KUKA KRL program: MyProgram_248().src

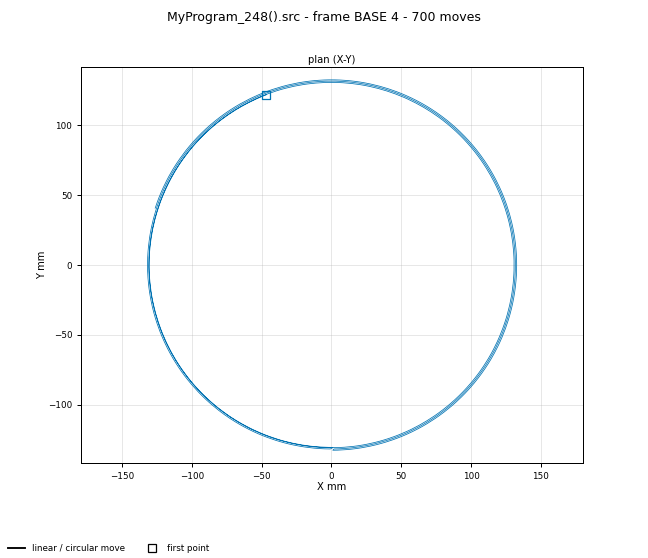
[picture p0: tool path of MyProgram_248().src in frame BASE 4, 700 of 700 moves have a stored position in this frame; points joined in program order, loops and branches not executed]
&ACCESS RVP
&REL 1
&PARAM TEMPLATE = C:\KRC\Roboter\Template\vorgabe
&PARAM EDITMASK = *
DEF MyProgram_248()
; ---- Setting reference (Base) ----
$BASE = BASE_DATA[4]

; --------------------------
; ---- Setting tool (TCP) ----
$TOOL = TOOL_DATA[3]
; --------------------------

$VEL.CP = VEL_APROX_PRINT
Startdeposition()
$VEL.CP = VEL_PRINT
LIN {X -46.6832,Y 121.9902,Z 163,A 110.8737,B 12.7153,C -0.1174,E1 12.6581,E2 699.2371} C_DIS
LIN {X -49.9782,Y 120.6763,Z 163,A 112.3319,B 12.7153,C -0.1132,E1 12.6544,E2 697.7915} C_DIS
LIN {X -53.5556,Y 119.1314,Z 163,A 114.1157,B 12.7153,C -0.1128,E1 12.6498,E2 696.0006} C_DIS
LIN {X -57.2848,Y 117.3848,Z 163,A 115.8599,B 12.7154,C -0.1089,E1 12.6454,E2 694.2652} C_DIS
LIN {X -59.7951,Y 116.1264,Z 163,A 117.1162,B 12.7154,C -0.1077,E1 12.6423,E2 693.0071} C_DIS
LIN {X -62.9383,Y 114.4547,Z 163,A 118.6303,B 12.7154,C -0.1043,E1 12.6386,E2 691.5001} C_DIS
LIN {X -65.207,Y 113.1772,Z 163,A 119.9528,B 12.7154,C -0.1069,E1 12.6353,E2 690.1578} C_DIS
LIN {X -68.5198,Y 111.2027,Z 163,A 121.5343,B 12.7154,C -0.1015,E1 12.6316,E2 688.5907} C_DIS
LIN {X -71.225,Y 109.4895,Z 163,A 122.9481,B 12.7155,C -0.0994,E1 12.6283,E2 687.1773} C_DIS
LIN {X -73.8707,Y 107.7222,Z 163,A 124.3516,B 12.7155,C -0.0972,E1 12.625,E2 685.7742} C_DIS
LIN {X -76.4904,Y 105.8783,Z 163,A 125.7574,B 12.7155,C -0.0947,E1 12.6218,E2 684.3698} C_DIS
LIN {X -79.0882,Y 103.9525,Z 163,A 127.1877,B 12.7155,C -0.0924,E1 12.6186,E2 682.9396} C_DIS
LIN {X -82.2352,Y 101.4811,Z 163,A 128.9913,B 12.7155,C -0.0902,E1 12.6147,E2 681.1323} C_DIS
LIN {X -85.3227,Y 98.8989,Z 163,A 130.775,B 12.7155,C -0.0871,E1 12.6109,E2 679.3484} C_DIS
LIN {X -88.3103,Y 96.2406,Z 163,A 132.6231,B 12.7156,C -0.0857,E1 12.607,E2 677.4913} C_DIS
LIN {X -91.2151,Y 93.4926,Z 163,A 134.4135,B 12.7156,C -0.0829,E1 12.6034,E2 675.6986} C_DIS
LIN {X -94.1515,Y 90.5351,Z 163,A 136.2687,B 12.7156,C -0.0795,E1 12.5998,E2 673.8423} C_DIS
LIN {X -97.2048,Y 87.2479,Z 163,A 138.1813,B 12.7156,C -0.0738,E1 12.5962,E2 671.9384} C_DIS
LIN {X -99.9408,Y 84.1001,Z 163,A 139.9545,B 12.7157,C -0.0683,E1 12.593,E2 670.1738} C_DIS
LIN {X -102.0114,Y 81.5764,Z 163,A 141.5514,B 12.7157,C -0.0687,E1 12.5902,E2 668.5594} C_DIS
LIN {X -104.7092,Y 78.083,Z 163,A 143.3581,B 12.7157,C -0.0611,E1 12.5872,E2 666.77} C_DIS
LIN {X -106.3801,Y 75.791,Z 163,A 144.7627,B 12.7157,C -0.0617,E1 12.5849,E2 665.3482} C_DIS
LIN {X -108.8838,Y 72.1487,Z 163,A 146.7321,B 12.7157,C -0.0576,E1 12.5818,E2 663.3776} C_DIS
LIN {X -111.0171,Y 68.8201,Z 163,A 148.3315,B 12.7157,C -0.05,E1 12.5794,E2 661.796} C_DIS
LIN {X -112.8395,Y 65.7903,Z 163,A 150.0583,B 12.7157,C -0.05,E1 12.5769,E2 660.0506} C_DIS
LIN {X -115.0342,Y 61.8715,Z 163,A 151.9693,B 12.7158,C -0.0435,E1 12.5744,E2 658.1488} C_DIS
LIN {X -116.6759,Y 58.7157,Z 163,A 153.4482,B 12.7158,C -0.0374,E1 12.5725,E2 656.6811} C_DIS
LIN {X -118.0782,Y 55.8412,Z 163,A 154.889,B 12.7158,C -0.0345,E1 12.5708,E2 655.2377} C_DIS
LIN {X -119.2704,Y 53.245,Z 163,A 156.2038,B 12.7158,C -0.0325,E1 12.5693,E2 653.9172} C_DIS
LIN {X -120.6709,Y 49.9913,Z 163,A 157.6764,B 12.7158,C -0.0263,E1 12.5677,E2 652.456} C_DIS
LIN {X -121.7339,Y 47.3425,Z 163,A 159.0481,B 12.7158,C -0.0256,E1 12.5663,E2 651.0717} C_DIS
LIN {X -122.9737,Y 44.023,Z 163,A 160.5652,B 12.7158,C -0.0203,E1 12.5648,E2 649.561} C_DIS
LIN {X -124.0232,Y 40.9732,Z 163,A 161.9931,B 12.7158,C -0.0166,E1 12.5635,E2 648.1332} C_DIS
LIN {X -124.9945,Y 37.9073,Z 163,A 163.4198,B 12.7158,C -0.0129,E1 12.5624,E2 646.7064} C_DIS
LIN {X -125.794,Y 35.1618,Z 163,A 164.7429,B 12.7158,C -0.0109,E1 12.5613,E2 645.3767} C_DIS
LIN {X -126.6177,Y 32.0694,Z 163,A 166.1098,B 12.7158,C -0.006,E1 12.5604,E2 644.0158} C_DIS
LIN {X -127.4419,Y 28.6231,Z 163,A 167.6781,B 12.7158,C -0.0018,E1 12.5594,E2 642.4477} C_DIS
LIN {X -128.0367,Y 25.8293,Z 163,A 168.986,B 12.7158,C 0.0007,E1 12.5587,E2 641.1349} C_DIS
LIN {X -128.6915,Y 22.3488,Z 163,A 170.4906,B 12.7158,C 0.0063,E1 12.5579,E2 639.6379} C_DIS
LIN {X -129.156,Y 19.4811,Z 163,A 171.8014,B 12.7158,C 0.0093,E1 12.5574,E2 638.3244} C_DIS
LIN {X -129.5892,Y 16.3576,Z 163,A 173.1987,B 12.7158,C 0.013,E1 12.5568,E2 636.927} C_DIS
LIN {X -129.9523,Y 13.1691,Z 163,A 174.7524,B 12.7158,C 0.0139,E1 12.5564,E2 635.3579} C_DIS
LIN {X -130.2342,Y 9.9928,Z 163,A 176.0604,B 12.7158,C 0.0201,E1 12.5561,E2 634.0621} C_DIS
LIN {X -130.4875,Y 5.8387,Z 163,A 178.0776,B 12.7158,C 0.0212,E1 12.5558,E2 632.0246} C_DIS
LIN {X -130.6007,Y 2.0177,Z 163,A 179.5385,B 12.7158,C 0.031,E1 12.5557,E2 630.5908} C_DIS
LIN {X -130.6106,Y -1.3842,Z 163,A -178.8919,B 12.7158,C 0.0337,E1 12.5557,E2 629.0138} C_DIS
LIN {X -130.52,Y -5.011,Z 163,A -177.2402,B 12.7158,C 0.037,E1 12.5559,E2 627.3568} C_DIS
LIN {X -130.3104,Y -8.9487,Z 163,A -175.3685,B 12.7158,C 0.0389,E1 12.5562,E2 625.4704} C_DIS
LIN {X -130.0173,Y -12.4916,Z 163,A -173.9505,B 12.7158,C 0.0467,E1 12.5565,E2 624.0706} C_DIS
LIN {X -129.633,Y -16.0033,Z 163,A -172.3925,B 12.7158,C 0.0511,E1 12.557,E2 622.5132} C_DIS
LIN {X -129.2325,Y -18.9667,Z 163,A -171.0719,B 12.7158,C 0.0547,E1 12.5575,E2 621.1929} C_DIS
LIN {X -128.8196,Y -21.5878,Z 163,A -169.825,B 12.7158,C 0.0562,E1 12.5581,E2 619.9375} C_DIS
LIN {X -128.1778,Y -25.1263,Z 163,A -168.2019,B 12.7158,C 0.0598,E1 12.559,E2 618.3106} C_DIS
LIN {X -127.5268,Y -28.2472,Z 163,A -166.7611,B 12.7158,C 0.0628,E1 12.5598,E2 616.8663} C_DIS
LIN {X -126.7017,Y -31.7385,Z 163,A -165.2684,B 12.7158,C 0.0692,E1 12.5608,E2 615.3846} C_DIS
LIN {X -125.9783,Y -34.5028,Z 163,A -164.042,B 12.7157,C 0.0733,E1 12.5617,E2 614.1626} C_DIS
LIN {X -125.0954,Y -37.5777,Z 163,A -162.5825,B 12.7157,C 0.076,E1 12.5628,E2 612.6978} C_DIS
LIN {X -124.1519,Y -40.5868,Z 163,A -161.1603,B 12.7157,C 0.079,E1 12.5641,E2 611.2723} C_DIS
LIN {X -123.0973,Y -43.6802,Z 163,A -159.7902,B 12.7157,C 0.0844,E1 12.5653,E2 609.9109} C_DIS
LIN {X -121.9894,Y -46.6852,Z 163,A -158.2103,B 12.7157,C 0.0842,E1 12.5669,E2 608.3117} C_DIS
LIN {X -120.672,Y -49.9886,Z 163,A -156.8729,B 12.7155,C 0.0936,E1 12.5683,E2 607.0018} C_DIS
LIN {X -119.4164,Y -52.9185,Z 163,A -155.3294,B 12.7155,C 0.0939,E1 12.57,E2 605.4423} C_DIS
LIN {X -118.2446,Y -55.4906,Z 163,A -153.9832,B 12.7155,C 0.0948,E1 12.5716,E2 604.0846} C_DIS
LIN {X -116.707,Y -58.6546,Z 163,A -152.5589,B 12.7155,C 0.1015,E1 12.5733,E2 602.6755} C_DIS
LIN {X -115.3567,Y -61.267,Z 163,A -151.1647,B 12.7155,C 0.1024,E1 12.5752,E2 601.27} C_DIS
LIN {X -113.82,Y -64.0779,Z 163,A -149.6509,B 12.7155,C 0.1034,E1 12.5772,E2 599.7444} C_DIS
LIN {X -111.5694,Y -67.9218,Z 163,A -147.6613,B 12.7155,C 0.1075,E1 12.5801,E2 597.7521} C_DIS
LIN {X -109.2975,Y -71.5202,Z 163,A -145.7821,B 12.7155,C 0.1117,E1 12.5829,E2 595.8727} C_DIS
LIN {X -106.7955,Y -75.2043,Z 163,A -144.0551,B 12.7153,C 0.1217,E1 12.5856,E2 594.1738} C_DIS
LIN {X -104.9142,Y -77.8076,Z 163,A -142.5374,B 12.7153,C 0.1224,E1 12.5881,E2 592.6441} C_DIS
LIN {X -103.0812,Y -80.2202,Z 163,A -141.1619,B 12.7153,C 0.1243,E1 12.5905,E2 591.2638} C_DIS
LIN {X -100.5659,Y -83.3513,Z 163,A -139.3096,B 12.7153,C 0.1261,E1 12.5938,E2 589.4018} C_DIS
LIN {X -97.7543,Y -86.6318,Z 163,A -137.3785,B 12.7153,C 0.1293,E1 12.5973,E2 587.4674} C_DIS
LIN {X -94.7689,Y -89.8884,Z 163,A -135.4961,B 12.7152,C 0.1347,E1 12.6009,E2 585.5926} C_DIS
LIN {X -91.916,Y -92.8033,Z 163,A -133.6849,B 12.7152,C 0.1377,E1 12.6045,E2 583.7796} C_DIS
LIN {X -88.9031,Y -95.6933,Z 163,A -131.769,B 12.7152,C 0.1393,E1 12.6084,E2 581.8544} C_DIS
LIN {X -85.9341,Y -98.3681,Z 163,A -130.0988,B 12.7151,C 0.1445,E1 12.6118,E2 580.1947} C_DIS
LIN {X -82.9209,Y -100.9217,Z 163,A -128.3556,B 12.7151,C 0.1474,E1 12.6156,E2 578.4509} C_DIS
LIN {X -79.8515,Y -103.367,Z 163,A -126.5261,B 12.7151,C 0.1477,E1 12.6196,E2 576.609} C_DIS
LIN {X -76.7991,Y -105.6545,Z 163,A -124.9687,B 12.715,C 0.1533,E1 12.6231,E2 575.0658} C_DIS
LIN {X -74.4284,Y -107.3378,Z 163,A -123.6386,B 12.715,C 0.154,E1 12.6262,E2 573.7295} C_DIS
LIN {X -72.0249,Y -108.9652,Z 163,A -122.2836,B 12.715,C 0.154,E1 12.6293,E2 572.3651} C_DIS
LIN {X -68.8174,Y -111.0188,Z 163,A -120.7144,B 12.715,C 0.1589,E1 12.633,E2 570.8084} C_DIS
LIN {X -66.0644,Y -112.6786,Z 163,A -119.3006,B 12.7149,C 0.1608,E1 12.6364,E2 569.3943} C_DIS
LIN {X -63.6337,Y -114.0696,Z 163,A -117.9724,B 12.7149,C 0.16,E1 12.6397,E2 568.0544} C_DIS
LIN {X -60.1614,Y -115.9372,Z 163,A -116.3208,B 12.7149,C 0.1641,E1 12.6437,E2 566.4122} C_DIS
LIN {X -57.6106,Y -117.2241,Z 163,A -115.0672,B 12.7149,C 0.1656,E1 12.6469,E2 565.1586} C_DIS
LIN {X -54.7716,Y -118.577,Z 163,A -113.6686,B 12.7149,C 0.1667,E1 12.6504,E2 563.7578} C_DIS
LIN {X -51.4577,Y -120.053,Z 163,A -112.082,B 12.7148,C 0.1685,E1 12.6545,E2 562.1718} C_DIS
LIN {X -48.8184,Y -121.1496,Z 163,A -110.8254,B 12.7148,C 0.1697,E1 12.6577,E2 560.9148} C_DIS
LIN {X -45.5127,Y -122.4302,Z 163,A -109.264,B 12.7148,C 0.171,E1 12.6618,E2 559.3526} C_DIS
LIN {X -42.4978,Y -123.5091,Z 163,A -107.8552,B 12.7148,C 0.172,E1 12.6655,E2 557.9432} C_DIS
LIN {X -39.4561,Y -124.5142,Z 163,A -106.4463,B 12.7148,C 0.1731,E1 12.6692,E2 556.5337} C_DIS
LIN {X -36.7579,Y -125.3369,Z 163,A -105.1944,B 12.7148,C 0.1736,E1 12.6726,E2 555.2799} C_DIS
LIN {X -33.3,Y -126.3002,Z 163,A -103.6737,B 12.7147,C 0.176,E1 12.6767,E2 553.7654} C_DIS
LIN {X -30.2058,Y -127.0759,Z 163,A -102.2279,B 12.7147,C 0.1756,E1 12.6806,E2 552.3137} C_DIS
LIN {X -27.1009,Y -127.7743,Z 163,A -100.8642,B 12.7147,C 0.1771,E1 12.6843,E2 550.9536} C_DIS
LIN {X -24.1906,Y -128.3567,Z 163,A -99.5117,B 12.7147,C 0.1763,E1 12.6881,E2 549.5946} C_DIS
LIN {X -21.085,Y -128.9035,Z 163,A -98.0994,B 12.7147,C 0.1761,E1 12.692,E2 548.1785} C_DIS
LIN {X -17.9213,Y -129.3819,Z 163,A -96.7699,B 12.7147,C 0.1784,E1 12.6956,E2 546.8575} C_DIS
LIN {X -14.7423,Y -129.7835,Z 163,A -95.212,B 12.7147,C 0.1747,E1 12.7,E2 545.2808} C_DIS
LIN {X -11.214,Y -130.134,Z 163,A -93.8584,B 12.7147,C 0.1802,E1 12.7037,E2 543.9507} C_DIS
LIN {X -8.366,Y -130.3483,Z 163,A -92.4343,B 12.7147,C 0.1758,E1 12.7077,E2 542.5055} C_DIS
LIN {X -5.153,Y -130.5145,Z 163,A -91.1022,B 12.7147,C 0.1779,E1 12.7114,E2 541.1823} C_DIS
LIN {X -1.9527,Y -130.6018,Z 163,A -89.6778,B 12.7147,C 0.1772,E1 12.7154,E2 539.7549} C_DIS
LIN {X 0.9174,Y -130.6131,Z 163,A -88.8333,B 12.7145,C 0.188,E1 12.7176,E2 538.9595} C_DIS
Enddeposition()
LIN {X 0.9174,Y -130.6131,Z 163,A -88.8333,B 12.7145,C 0.188,E1 12.7176,E2 538.9595} C_DIS
Startdeposition()
$VEL.CP = VEL_PRINT
LIN {X 2.9572,Y -130.8103,Z 164,A -87.5272,B 12.7129,C 0.1767,E1 12.7196,E2 537.6024} C_DIS
LIN {X 6.1659,Y -130.6972,Z 164,A -86.0767,B 12.7129,C 0.1751,E1 12.7236,E2 536.1458} C_DIS
LIN {X 9.3838,Y -130.505,Z 164,A -84.7313,B 12.7129,C 0.1764,E1 12.7274,E2 534.8076} C_DIS
LIN {X 12.8176,Y -130.2129,Z 164,A -83.2362,B 12.7129,C 0.1762,E1 12.7315,E2 533.3133} C_DIS
LIN {X 15.6281,Y -129.9052,Z 164,A -81.9766,B 12.7129,C 0.175,E1 12.735,E2 532.0504} C_DIS
LIN {X 18.9476,Y -129.4633,Z 164,A -80.5189,B 12.7129,C 0.1744,E1 12.739,E2 530.5928} C_DIS
LIN {X 22.132,Y -128.9577,Z 164,A -79.0774,B 12.7129,C 0.1727,E1 12.743,E2 529.1468} C_DIS
LIN {X 25.5213,Y -128.3298,Z 164,A -77.6997,B 12.7129,C 0.1753,E1 12.7468,E2 527.784} C_DIS
LIN {X 28.6831,Y -127.6598,Z 164,A -76.2844,B 12.7129,C 0.1742,E1 12.7506,E2 526.3676} C_DIS
LIN {X 30.9937,Y -127.1182,Z 164,A -75.149,B 12.7129,C 0.1707,E1 12.7538,E2 525.2199} C_DIS
LIN {X 34.8731,Y -126.1092,Z 164,A -73.5047,B 12.7129,C 0.1721,E1 12.7582,E2 523.5877} C_DIS
LIN {X 37.9309,Y -125.2234,Z 164,A -72.07,B 12.7129,C 0.1697,E1 12.762,E2 522.147} C_DIS
LIN {X 41.2594,Y -124.1659,Z 164,A -70.4025,B 12.713,C 0.1643,E1 12.7665,E2 520.4615} C_DIS
LIN {X 45.586,Y -122.6438,Z 164,A -68.5096,B 12.713,C 0.1652,E1 12.7714,E2 518.5809} C_DIS
LIN {X 48.3557,Y -121.5795,Z 164,A -67.2192,B 12.713,C 0.1639,E1 12.7748,E2 517.2906} C_DIS
LIN {X 51.5406,Y -120.2631,Z 164,A -65.8052,B 12.713,C 0.1646,E1 12.7784,E2 515.8866} C_DIS
LIN {X 54.2495,Y -119.0672,Z 164,A -64.4511,B 12.713,C 0.1612,E1 12.7819,E2 514.5245} C_DIS
LIN {X 57.1852,Y -117.6857,Z 164,A -63.0198,B 12.713,C 0.1589,E1 12.7855,E2 513.0907} C_DIS
LIN {X 60.261,Y -116.1399,Z 164,A -61.5367,B 12.7131,C 0.1574,E1 12.7892,E2 511.609} C_DIS
LIN {X 62.8821,Y -114.7428,Z 164,A -60.1838,B 12.7131,C 0.1539,E1 12.7925,E2 510.2486} C_DIS
LIN {X 65.678,Y -113.1654,Z 164,A -58.8716,B 12.7131,C 0.1543,E1 12.7957,E2 508.9464} C_DIS
LIN {X 68.4316,Y -111.5218,Z 164,A -57.43,B 12.7131,C 0.1509,E1 12.7991,E2 507.4988} C_DIS
LIN {X 71.1439,Y -109.8114,Z 164,A -56.0328,B 12.7132,C 0.1487,E1 12.8024,E2 506.101} C_DIS
LIN {X 73.8295,Y -108.0243,Z 164,A -54.6378,B 12.7132,C 0.1467,E1 12.8056,E2 504.7068} C_DIS
LIN {X 76.4534,Y -106.1839,Z 164,A -53.1819,B 12.7132,C 0.1427,E1 12.809,E2 503.2431} C_DIS
LIN {X 79.7631,Y -103.7205,Z 164,A -51.426,B 12.7132,C 0.1407,E1 12.8129,E2 501.4913} C_DIS
LIN {X 82.9013,Y -101.2293,Z 164,A -49.6993,B 12.7133,C 0.138,E1 12.8166,E2 499.7662} C_DIS
LIN {X 85.3739,Y -99.1528,Z 164,A -48.2801,B 12.7133,C 0.135,E1 12.8197,E2 498.3448} C_DIS
LIN {X 88.3689,Y -96.4934,Z 164,A -46.5394,B 12.7133,C 0.1317,E1 12.8233,E2 496.6037} C_DIS
LIN {X 91.3657,Y -93.6612,Z 164,A -44.7492,B 12.7134,C 0.1283,E1 12.8269,E2 494.8134} C_DIS
LIN {X 94.2093,Y -90.8002,Z 164,A -42.8838,B 12.7134,C 0.1215,E1 12.8305,E2 492.9339} C_DIS
LIN {X 97.0246,Y -87.7852,Z 164,A -41.0985,B 12.7135,C 0.118,E1 12.8339,E2 491.1491} C_DIS
LIN {X 100.0304,Y -84.3446,Z 164,A -39.2261,B 12.7135,C 0.117,E1 12.8373,E2 489.2899} C_DIS
LIN {X 102.5806,Y -81.2238,Z 164,A -37.4588,B 12.7135,C 0.1127,E1 12.8404,E2 487.5203} C_DIS
LIN {X 105.0905,Y -77.9488,Z 164,A -35.7098,B 12.7135,C 0.11,E1 12.8433,E2 485.776} C_DIS
LIN {X 106.8866,Y -75.4668,Z 164,A -34.3578,B 12.7136,C 0.1063,E1 12.8455,E2 484.4212} C_DIS
LIN {X 108.7849,Y -72.7038,Z 164,A -32.9309,B 12.7136,C 0.1038,E1 12.8478,E2 482.9975} C_DIS
LIN {X 110.5434,Y -70.0013,Z 164,A -31.5399,B 12.7136,C 0.1008,E1 12.8499,E2 481.6073} C_DIS
LIN {X 112.2262,Y -67.2709,Z 164,A -29.9994,B 12.7137,C 0.0932,E1 12.8521,E2 480.0487} C_DIS
LIN {X 114.5187,Y -63.2888,Z 164,A -28.1177,B 12.7137,C 0.0917,E1 12.8547,E2 478.1804} C_DIS
LIN {X 116.0276,Y -60.4749,Z 164,A -26.7681,B 12.7137,C 0.0893,E1 12.8564,E2 476.8349} C_DIS
LIN {X 117.5747,Y -57.4102,Z 164,A -25.2801,B 12.7137,C 0.0857,E1 12.8583,E2 475.3468} C_DIS
LIN {X 118.8392,Y -54.7426,Z 164,A -23.9675,B 12.7138,C 0.0815,E1 12.8598,E2 474.0303} C_DIS
LIN {X 120.259,Y -51.5502,Z 164,A -22.5189,B 12.7138,C 0.0797,E1 12.8614,E2 472.5896} C_DIS
LIN {X 121.4863,Y -48.5868,Z 164,A -21.1028,B 12.7138,C 0.0754,E1 12.8629,E2 471.1704} C_DIS
LIN {X 122.5606,Y -45.8082,Z 164,A -19.7787,B 12.7138,C 0.0712,E1 12.8642,E2 469.8424} C_DIS
LIN {X 123.9688,Y -41.8512,Z 164,A -17.8515,B 12.7139,C 0.0633,E1 12.866,E2 467.9023} C_DIS
LIN {X 125.1387,Y -38.2075,Z 164,A -16.3407,B 12.7139,C 0.0633,E1 12.8673,E2 466.4094} C_DIS
LIN {X 126.1006,Y -34.9037,Z 164,A -14.8825,B 12.7139,C 0.0605,E1 12.8684,E2 464.9552} C_DIS
LIN {X 126.9173,Y -31.807,Z 164,A -13.468,B 12.7139,C 0.056,E1 12.8694,E2 463.5376} C_DIS
LIN {X 127.6574,Y -28.6936,Z 164,A -12.1068,B 12.7139,C 0.0531,E1 12.8702,E2 462.1795} C_DIS
LIN {X 128.3029,Y -25.6535,Z 164,A -10.7502,B 12.7139,C 0.0492,E1 12.871,E2 460.8218} C_DIS
LIN {X 128.8767,Y -22.5953,Z 164,A -9.3815,B 12.7139,C 0.045,E1 12.8717,E2 459.4507} C_DIS
LIN {X 129.3921,Y -19.4319,Z 164,A -7.9572,B 12.7139,C 0.0403,E1 12.8723,E2 458.0224} C_DIS
LIN {X 129.8586,Y -16.0182,Z 164,A -6.4988,B 12.714,C 0.0373,E1 12.8728,E2 456.5682} C_DIS
LIN {X 130.1891,Y -13.0648,Z 164,A -5.212,B 12.714,C 0.0339,E1 12.8732,E2 455.2816} C_DIS
LIN {X 130.487,Y -9.63,Z 164,A -3.7393,B 12.714,C 0.0305,E1 12.8735,E2 453.8116} C_DIS
LIN {X 130.6726,Y -6.6548,Z 164,A -2.4043,B 12.714,C 0.0257,E1 12.8737,E2 452.4715} C_DIS
LIN {X 130.7933,Y -3.5686,Z 164,A -1.0691,B 12.714,C 0.0222,E1 12.8738,E2 451.1369} C_DIS
LIN {X 130.8438,Y -0.0051,Z 164,A 0.3845,B 12.714,C 0.0207,E1 12.8738,E2 449.6944} C_DIS
LIN {X 130.81,Y 2.965,Z 164,A 1.7444,B 12.714,C 0.0151,E1 12.8738,E2 448.3259} C_DIS
LIN {X 130.7112,Y 5.8858,Z 164,A 3.1328,B 12.714,C 0.0081,E1 12.8736,E2 446.9232} C_DIS
LIN {X 130.5047,Y 9.3874,Z 164,A 4.5066,B 12.714,C 0.0083,E1 12.8734,E2 445.5671} C_DIS
LIN {X 130.2123,Y 12.8233,Z 164,A 5.9871,B 12.714,C 0.0047,E1 12.873,E2 444.0885} C_DIS
LIN {X 129.8877,Y 15.7743,Z 164,A 7.2744,B 12.714,C 0.0013,E1 12.8726,E2 442.8013} C_DIS
LIN {X 129.4605,Y 18.9672,Z 164,A 8.6844,B 12.714,C -0.0028,E1 12.872,E2 441.3899} C_DIS
LIN {X 128.9575,Y 22.1333,Z 164,A 10.0542,B 12.714,C -0.0059,E1 12.8714,E2 440.0228} C_DIS
LIN {X 128.3296,Y 25.5223,Z 164,A 11.4734,B 12.714,C -0.0077,E1 12.8707,E2 438.6127} C_DIS
LIN {X 127.6647,Y 28.6616,Z 164,A 12.8714,B 12.714,C -0.0115,E1 12.8698,E2 437.2142} C_DIS
LIN {X 127.1257,Y 30.9627,Z 164,A 14.0476,B 12.714,C -0.0186,E1 12.8691,E2 436.0201} C_DIS
LIN {X 126.1183,Y 34.8406,Z 164,A 15.5966,B 12.714,C -0.0176,E1 12.868,E2 434.4939} C_DIS
LIN {X 125.2532,Y 37.8335,Z 164,A 17.002,B 12.714,C -0.0226,E1 12.8668,E2 433.0824} C_DIS
LIN {X 124.4586,Y 40.372,Z 164,A 18.3592,B 12.714,C -0.0315,E1 12.8657,E2 431.7012} C_DIS
LIN {X 123.194,Y 44.0777,Z 164,A 19.896,B 12.714,C -0.0311,E1 12.8643,E2 430.184} C_DIS
LIN {X 122.0769,Y 47.0833,Z 164,A 21.2033,B 12.714,C -0.0321,E1 12.863,E2 428.887} C_DIS
LIN {X 120.9801,Y 49.8367,Z 164,A 22.5072,B 12.714,C -0.0358,E1 12.8616,E2 427.5813} C_DIS
LIN {X 119.7152,Y 52.8035,Z 164,A 23.9618,B 12.714,C -0.0409,E1 12.86,E2 426.1206} C_DIS
LIN {X 118.4142,Y 55.6615,Z 164,A 25.3445,B 12.714,C -0.0447,E1 12.8584,E2 424.7359} C_DIS
LIN {X 116.9748,Y 58.6262,Z 164,A 26.8279,B 12.714,C -0.0497,E1 12.8565,E2 423.2465} C_DIS
LIN {X 115.3941,Y 61.6787,Z 164,A 28.1997,B 12.714,C -0.0497,E1 12.8548,E2 421.8894} C_DIS
LIN {X 114.0584,Y 64.1144,Z 164,A 29.4816,B 12.714,C -0.0547,E1 12.853,E2 420.5988} C_DIS
LIN {X 112.3615,Y 67.044,Z 164,A 30.9152,B 12.714,C -0.057,E1 12.851,E2 419.1699} C_DIS
LIN {X 110.8493,Y 69.5166,Z 164,A 32.2505,B 12.714,C -0.0621,E1 12.849,E2 417.8259} C_DIS
LIN {X 108.9256,Y 72.493,Z 164,A 33.7051,B 12.714,C -0.0631,E1 12.8468,E2 416.3818} C_DIS
LIN {X 107.1096,Y 75.1506,Z 164,A 35.0977,B 12.7139,C -0.066,E1 12.8446,E2 414.9902} C_DIS
LIN {X 105.0942,Y 77.9439,Z 164,A 36.7258,B 12.7139,C -0.0729,E1 12.8419,E2 413.3471} C_DIS
LIN {X 102.6588,Y 81.1252,Z 164,A 38.4806,B 12.7139,C -0.0769,E1 12.8389,E2 411.5912} C_DIS
LIN {X 100.2025,Y 84.1395,Z 164,A 40.0666,B 12.7139,C -0.0774,E1 12.836,E2 410.0181} C_DIS
LIN {X 97.4808,Y 87.2782,Z 164,A 41.9544,B 12.7138,C -0.0833,E1 12.8325,E2 408.1212} C_DIS
LIN {X 94.7615,Y 90.2236,Z 164,A 43.696,B 12.7138,C -0.0866,E1 12.8292,E2 406.3804} C_DIS
LIN {X 91.9519,Y 93.0858,Z 164,A 45.4537,B 12.7138,C -0.0903,E1 12.8257,E2 404.6217} C_DIS
LIN {X 88.9689,Y 95.9406,Z 164,A 47.2429,B 12.7138,C -0.0933,E1 12.8221,E2 402.834} C_DIS
LIN {X 85.7549,Y 98.8241,Z 164,A 49.0357,B 12.7138,C -0.0942,E1 12.8184,E2 401.0521} C_DIS
LIN {X 82.9996,Y 101.149,Z 164,A 50.6759,B 12.7137,C -0.0988,E1 12.8148,E2 399.404} C_DIS
LIN {X 79.7682,Y 103.7166,Z 164,A 52.4795,B 12.7137,C -0.1019,E1 12.8109,E2 397.6004} C_DIS
LIN {X 76.6517,Y 106.0402,Z 164,A 54.0346,B 12.7137,C -0.1007,E1 12.8074,E2 396.0621} C_DIS
LIN {X 74.0284,Y 107.8878,Z 164,A 55.3783,B 12.7137,C -0.1013,E1 12.8043,E2 394.7252} C_DIS
LIN {X 71.3742,Y 109.6619,Z 164,A 56.8102,B 12.7137,C -0.1044,E1 12.801,E2 393.289} C_DIS
LIN {X 68.6418,Y 111.3928,Z 164,A 58.2207,B 12.7137,C -0.1064,E1 12.7976,E2 391.8789} C_DIS
LIN {X 65.8901,Y 113.0426,Z 164,A 59.6239,B 12.7137,C -0.1084,E1 12.7943,E2 390.4758} C_DIS
LIN {X 63.2961,Y 114.5146,Z 164,A 60.9593,B 12.7136,C -0.111,E1 12.791,E2 389.1367} C_DIS
LIN {X 60.4719,Y 116.0292,Z 164,A 62.3206,B 12.7136,C -0.1117,E1 12.7877,E2 387.7801} C_DIS
LIN {X 57.3978,Y 117.5808,Z 164,A 63.7226,B 12.7136,C -0.1107,E1 12.7842,E2 386.3904} C_DIS
LIN {X 54.7508,Y 118.8354,Z 164,A 65.1214,B 12.7136,C -0.1154,E1 12.7806,E2 384.9779} C_DIS
LIN {X 51.8699,Y 120.1207,Z 164,A 66.4869,B 12.7136,C -0.1165,E1 12.7771,E2 383.6143} C_DIS
LIN {X 48.5905,Y 121.4848,Z 164,A 68.0197,B 12.7136,C -0.1176,E1 12.7732,E2 382.0842} C_DIS
LIN {X 45.8111,Y 122.5595,Z 164,A 69.3167,B 12.7136,C -0.1186,E1 12.7698,E2 380.7881} C_DIS
LIN {X 42.7934,Y 123.6456,Z 164,A 70.7158,B 12.7136,C -0.1198,E1 12.7661,E2 379.3898} C_DIS
LIN {X 39.7502,Y 124.6572,Z 164,A 72.115,B 12.7135,C -0.1209,E1 12.7624,E2 377.9913} C_DIS
LIN {X 36.6835,Y 125.5939,Z 164,A 73.5501,B 12.7135,C -0.1228,E1 12.7585,E2 376.5528} C_DIS
LIN {X 33.5741,Y 126.4607,Z 164,A 74.9551,B 12.7135,C -0.1235,E1 12.7547,E2 375.1489} C_DIS
LIN {X 30.241,Y 127.2996,Z 164,A 76.4213,B 12.7135,C -0.1235,E1 12.7508,E2 373.6877} C_DIS
LIN {X 27.3545,Y 127.9505,Z 164,A 77.6363,B 12.7135,C -0.1221,E1 12.7475,E2 372.4823} C_DIS
LIN {X 24.1889,Y 128.5869,Z 164,A 79.1239,B 12.7135,C -0.1247,E1 12.7434,E2 370.9864} C_DIS
LIN {X 20.7945,Y 129.1809,Z 164,A 80.6212,B 12.7135,C -0.125,E1 12.7393,E2 369.4911} C_DIS
LIN {X 17.6069,Y 129.6532,Z 164,A 82.0569,B 12.7135,C -0.1262,E1 12.7353,E2 368.0529} C_DIS
LIN {X 14.4223,Y 130.0452,Z 164,A 83.3824,B 12.7135,C -0.1245,E1 12.7316,E2 366.737} C_DIS
LIN {X 11.4698,Y 130.3389,Z 164,A 84.8155,B 12.7135,C -0.1283,E1 12.7276,E2 365.2889} C_DIS
LIN {X 8.2902,Y 130.5792,Z 164,A 86.1529,B 12.7135,C -0.1269,E1 12.7239,E2 363.9589} C_DIS
LIN {X 5.0188,Y 130.7457,Z 164,A 87.5978,B 12.7135,C -0.1273,E1 12.7199,E2 362.5133} C_DIS
LIN {X 1.6085,Y 130.8333,Z 164,A 89.0368,B 12.7135,C -0.1258,E1 12.7159,E2 361.0814} C_DIS
LIN {X -1.5992,Y 130.8335,Z 164,A 90.4132,B 12.7135,C -0.125,E1 12.7121,E2 359.709} C_DIS
LIN {X -4.5697,Y 130.7632,Z 164,A 91.7931,B 12.7135,C -0.1268,E1 12.7082,E2 358.3206} C_DIS
LIN {X -8.0118,Y 130.5964,Z 164,A 93.1603,B 12.7135,C -0.1229,E1 12.7044,E2 356.9706} C_DIS
LIN {X -10.9858,Y 130.3798,Z 164,A 94.6327,B 12.7135,C -0.1267,E1 12.7003,E2 355.4796} C_DIS
LIN {X -14.4179,Y 130.0457,Z 164,A 96.0767,B 12.7135,C -0.1245,E1 12.6963,E2 354.0441} C_DIS
LIN {X -17.363,Y 129.6851,Z 164,A 97.4026,B 12.7135,C -0.1245,E1 12.6926,E2 352.7159} C_DIS
LIN {X -20.3979,Y 129.2425,Z 164,A 98.7623,B 12.7135,C -0.1243,E1 12.6888,E2 351.3551} C_DIS
LIN {X -23.9457,Y 128.6334,Z 164,A 100.3542,B 12.7135,C -0.1237,E1 12.6845,E2 349.7625} C_DIS
LIN {X -26.8902,Y 128.0508,Z 164,A 101.7345,B 12.7135,C -0.1245,E1 12.6807,E2 348.3755} C_DIS
LIN {X -30.0123,Y 127.3548,Z 164,A 103.0636,B 12.7135,C -0.1217,E1 12.6771,E2 347.0557} C_DIS
LIN {X -33.1186,Y 126.5822,Z 164,A 104.539,B 12.7135,C -0.1224,E1 12.6731,E2 345.5727} C_DIS
LIN {X -36.2059,Y 125.7338,Z 164,A 105.944,B 12.7135,C -0.1212,E1 12.6693,E2 344.1683} C_DIS
LIN {X -39.5018,Y 124.7366,Z 164,A 107.3859,B 12.7135,C -0.1182,E1 12.6655,E2 342.7353} C_DIS
LIN {X -42.5426,Y 123.7325,Z 164,A 108.7995,B 12.7135,C -0.1171,E1 12.6617,E2 341.3215} C_DIS
LIN {X -45.4393,Y 122.6988,Z 164,A 110.1922,B 12.7135,C -0.1167,E1 12.6581,E2 339.9246} C_DIS
LIN {X -48.3601,Y 121.5777,Z 164,A 111.5195,B 12.7135,C -0.1141,E1 12.6546,E2 338.6035} C_DIS
LIN {X -51.1469,Y 120.4329,Z 164,A 112.9042,B 12.7135,C -0.1141,E1 12.651,E2 337.2122} C_DIS
LIN {X -54.2864,Y 119.0501,Z 164,A 114.4294,B 12.7135,C -0.1127,E1 12.6472,E2 335.6857} C_DIS
LIN {X -57.1797,Y 117.6884,Z 164,A 115.7611,B 12.7135,C -0.1092,E1 12.6438,E2 334.3633} C_DIS
LIN {X -60.2505,Y 116.1454,Z 164,A 117.2562,B 12.7136,C -0.1068,E1 12.6401,E2 332.8706} C_DIS
LIN {X -62.8599,Y 114.7548,Z 164,A 118.6178,B 12.7136,C -0.1065,E1 12.6368,E2 331.5026} C_DIS
LIN {X -65.6417,Y 113.1864,Z 164,A 119.9905,B 12.7136,C -0.1037,E1 12.6334,E2 330.1342} C_DIS
LIN {X -68.3777,Y 111.5548,Z 164,A 121.2822,B 12.7136,C -0.099,E1 12.6304,E2 328.8558} C_DIS
LIN {X -70.7876,Y 110.0417,Z 164,A 122.7415,B 12.7136,C -0.1021,E1 12.6269,E2 327.373} C_DIS
LIN {X -73.8298,Y 108.0241,Z 164,A 124.2531,B 12.7136,C -0.0973,E1 12.6234,E2 325.8731} C_DIS
LIN {X -76.453,Y 106.1842,Z 164,A 125.7318,B 12.7136,C -0.0966,E1 12.62,E2 324.387} C_DIS
LIN {X -79.7555,Y 103.7264,Z 164,A 127.5115,B 12.7137,C -0.0927,E1 12.6161,E2 322.6119} C_DIS
LIN {X -82.9065,Y 101.2251,Z 164,A 129.2696,B 12.7137,C -0.0892,E1 12.6123,E2 320.8561} C_DIS
LIN {X -85.3748,Y 99.152,Z 164,A 130.7112,B 12.7137,C -0.0871,E1 12.6092,E2 319.4126} C_DIS
LIN {X -88.3717,Y 96.4908,Z 164,A 132.5101,B 12.7137,C -0.0846,E1 12.6054,E2 317.6104} C_DIS
LIN {X -91.3716,Y 93.6554,Z 164,A 134.3068,B 12.7138,C -0.0805,E1 12.6018,E2 315.817} C_DIS
LIN {X -94.2095,Y 90.8,Z 164,A 136.2019,B 12.7138,C -0.0798,E1 12.5981,E2 313.9085} C_DIS
LIN {X -96.9464,Y 87.8713,Z 164,A 137.964,B 12.7138,C -0.076,E1 12.5948,E2 312.1476} C_DIS
LIN {X -99.7376,Y 84.69,Z 164,A 139.8101,B 12.7138,C -0.0716,E1 12.5914,E2 310.3044} C_DIS
LIN {X -102.5815,Y 81.2227,Z 164,A 141.7301,B 12.7138,C -0.0659,E1 12.5881,E2 308.3918} C_DIS
LIN {X -105.0931,Y 77.9454,Z 164,A 143.5149,B 12.7139,C -0.061,E1 12.5851,E2 306.6119} C_DIS
LIN {X -106.9728,Y 75.3447,Z 164,A 144.9031,B 12.7139,C -0.0572,E1 12.5828,E2 305.2272} C_DIS
LIN {X -108.7823,Y 72.7076,Z 164,A 146.3363,B 12.7139,C -0.0544,E1 12.5806,E2 303.7919} C_DIS
LIN {X -110.5227,Y 70.0341,Z 164,A 147.7441,B 12.7139,C -0.0511,E1 12.5785,E2 302.3846} C_DIS
LIN {X -112.1704,Y 67.3643,Z 164,A 149.144,B 12.7139,C -0.0482,E1 12.5764,E2 300.9833} C_DIS
LIN {X -113.7026,Y 64.7435,Z 164,A 150.5001,B 12.7139,C -0.0453,E1 12.5745,E2 299.6257} C_DIS
LIN {X -115.3943,Y 61.6784,Z 164,A 152.0503,B 12.7139,C -0.0416,E1 12.5725,E2 298.0753} C_DIS
LIN {X -116.7622,Y 59.0439,Z 164,A 153.3811,B 12.714,C -0.0389,E1 12.5708,E2 296.7424} C_DIS
LIN {X -118.1682,Y 56.1766,Z 164,A 154.7719,B 12.714,C -0.0349,E1 12.5691,E2 295.3542} C_DIS
LIN {X -119.6142,Y 53.0293,Z 164,A 156.3032,B 12.714,C -0.0311,E1 12.5673,E2 293.823} C_DIS
LIN {X -120.7829,Y 50.3089,Z 164,A 157.7452,B 12.714,C -0.0308,E1 12.5658,E2 292.3656} C_DIS
LIN {X -122.5626,Y 45.8029,Z 164,A 159.7582,B 12.714,C -0.0224,E1 12.5637,E2 290.3678} C_DIS
LIN {X -123.6484,Y 42.7852,Z 164,A 161.1784,B 12.714,C -0.0188,E1 12.5624,E2 288.9475} C_DIS
LIN {X -124.66,Y 39.7415,Z 164,A 162.5992,B 12.714,C -0.0152,E1 12.5612,E2 287.5264} C_DIS
LIN {X -125.5974,Y 36.6719,Z 164,A 164.0562,B 12.714,C -0.0123,E1 12.56,E2 286.0652} C_DIS
LIN {X -126.458,Y 33.5846,Z 164,A 165.4741,B 12.714,C -0.0086,E1 12.559,E2 284.6472} C_DIS
LIN {X -127.2991,Y 30.2431,Z 164,A 166.9646,B 12.714,C -0.0038,E1 12.558,E2 283.1608} C_DIS
LIN {X -127.9567,Y 27.3258,Z 164,A 168.314,B 12.714,C -0.0009,E1 12.5572,E2 281.8082} C_DIS
LIN {X -128.5869,Y 24.189,Z 164,A 169.7055,B 12.714,C 0.0035,E1 12.5565,E2 280.4194} C_DIS
LIN {X -129.179,Y 20.8059,Z 164,A 171.2185,B 12.714,C 0.0077,E1 12.5558,E2 278.9072} C_DIS
LIN {X -129.6483,Y 17.6436,Z 164,A 172.6627,B 12.714,C 0.0108,E1 12.5552,E2 277.4595} C_DIS
LIN {X -130.0398,Y 14.4725,Z 164,A 173.9868,B 12.714,C 0.0167,E1 12.5548,E2 276.1457} C_DIS
LIN {X -130.3401,Y 11.4558,Z 164,A 175.4781,B 12.714,C 0.0169,E1 12.5544,E2 274.6368} C_DIS
LIN {X -130.5958,Y 8.0206,Z 164,A 176.8894,B 12.714,C 0.0235,E1 12.5541,E2 273.2386} C_DIS
LIN {X -130.7333,Y 5.3344,Z 164,A 178.2219,B 12.714,C 0.0235,E1 12.5539,E2 271.8894} C_DIS
LIN {X -130.8333,Y 1.6097,Z 164,A 179.7634,B 12.714,C 0.0304,E1 12.5539,E2 270.3603} C_DIS
LIN {X -130.8372,Y -1.2667,Z 164,A -178.929,B 12.714,C 0.0331,E1 12.5539,E2 269.0485} C_DIS
LIN {X -130.7627,Y -4.5829,Z 164,A -177.4579,B 12.714,C 0.0369,E1 12.5539,E2 267.5767} C_DIS
LIN {X -130.5956,Y -8.0243,Z 164,A -175.9946,B 12.714,C 0.0424,E1 12.5542,E2 266.1204} C_DIS
LIN {X -130.3797,Y -10.9875,Z 164,A -174.5916,B 12.714,C 0.044,E1 12.5545,E2 264.7068} C_DIS
LIN {X -129.9621,Y -15.1508,Z 164,A -172.6626,B 12.714,C 0.0471,E1 12.5551,E2 262.7684} C_DIS
LIN {X -129.4928,Y -18.7415,Z 164,A -171.1847,B 12.714,C 0.0542,E1 12.5557,E2 261.3048} C_DIS
LIN {X -128.9572,Y -22.1353,Z 164,A -169.6034,B 12.714,C 0.0569,E1 12.5564,E2 259.7161} C_DIS
LIN {X -128.3319,Y -25.511,Z 164,A -168.2089,B 12.714,C 0.0637,E1 12.5571,E2 258.3359} C_DIS
LIN {X -127.6632,Y -28.6684,Z 164,A -166.776,B 12.7139,C 0.0673,E1 12.558,E2 256.9021} C_DIS
LIN {X -127.0764,Y -31.1671,Z 164,A -165.4907,B 12.7139,C 0.0668,E1 12.5588,E2 255.5989} C_DIS
LIN {X -126.1056,Y -34.886,Z 164,A -163.9346,B 12.7139,C 0.0745,E1 12.5599,E2 254.0594} C_DIS
LIN {X -125.2134,Y -37.9634,Z 164,A -162.4283,B 12.7139,C 0.0761,E1 12.5611,E2 252.5422} C_DIS
LIN {X -124.2387,Y -41.0408,Z 164,A -161.0053,B 12.7139,C 0.0798,E1 12.5624,E2 251.1194} C_DIS
LIN {X -123.195,Y -44.0747,Z 164,A -159.4472,B 12.7139,C 0.0802,E1 12.5638,E2 249.5445} C_DIS
LIN {X -121.5814,Y -48.351,Z 164,A -157.5592,B 12.7138,C 0.0883,E1 12.5657,E2 247.6717} C_DIS
LIN {X -120.2957,Y -51.4653,Z 164,A -156.122,B 12.7138,C 0.0931,E1 12.5673,E2 246.2402} C_DIS
LIN {X -119.129,Y -54.1141,Z 164,A -154.6778,B 12.7138,C 0.0924,E1 12.5689,E2 244.7762} C_DIS
LIN {X -117.7013,Y -57.1535,Z 164,A -153.2962,B 12.7137,C 0.0983,E1 12.5706,E2 243.4063} C_DIS
LIN {X -116.1429,Y -60.2553,Z 164,A -151.7892,B 12.7137,C 0.1025,E1 12.5725,E2 241.902} C_DIS
LIN {X -114.7474,Y -62.8735,Z 164,A -150.4554,B 12.7137,C 0.1051,E1 12.5743,E2 240.565} C_DIS
LIN {X -113.1728,Y -65.6652,Z 164,A -149.0327,B 12.7137,C 0.1081,E1 12.5762,E2 239.1412} C_DIS
LIN {X -111.5185,Y -68.437,Z 164,A -147.6589,B 12.7136,C 0.1126,E1 12.5782,E2 237.773} C_DIS
LIN {X -109.8039,Y -71.1554,Z 164,A -146.2156,B 12.7136,C 0.1152,E1 12.5804,E2 236.3265} C_DIS
LIN {X -108.033,Y -73.8169,Z 164,A -144.7787,B 12.7136,C 0.1176,E1 12.5827,E2 234.8861} C_DIS
LIN {X -106.1827,Y -76.4551,Z 164,A -143.2884,B 12.7136,C 0.1191,E1 12.5851,E2 233.3873} C_DIS
LIN {X -103.719,Y -79.7651,Z 164,A -141.502,B 12.7135,C 0.1237,E1 12.5881,E2 231.6044} C_DIS
LIN {X -101.2262,Y -82.9051,Z 164,A -139.7193,B 12.7135,C 0.127,E1 12.5912,E2 229.8196} C_DIS
LIN {X -99.0964,Y -85.4394,Z 164,A -138.1648,B 12.7135,C 0.1276,E1 12.594,E2 228.2533} C_DIS
LIN {X -96.4834,Y -88.3798,Z 164,A -136.4232,B 12.7134,C 0.1308,E1 12.5973,E2 226.5104} C_DIS
LIN {X -93.6505,Y -91.3766,Z 164,A -134.7034,B 12.7134,C 0.1366,E1 12.6006,E2 224.8017} C_DIS
LIN {X -90.8049,Y -94.2047,Z 164,A -132.8165,B 12.7134,C 0.1369,E1 12.6044,E2 222.9} C_DIS
LIN {X -87.8941,Y -96.9258,Z 164,A -131.0652,B 12.7133,C 0.1401,E1 12.608,E2 221.1487} C_DIS
LIN {X -84.8891,Y -99.5684,Z 164,A -129.2949,B 12.7133,C 0.1429,E1 12.6118,E2 219.3769} C_DIS
LIN {X -81.375,Y -102.4603,Z 164,A -127.3522,B 12.7133,C 0.1476,E1 12.616,E2 217.4408} C_DIS
LIN {X -77.9488,Y -105.0905,Z 164,A -125.5387,B 12.7132,C 0.1527,E1 12.62,E2 215.6372} C_DIS
LIN {X -75.3444,Y -106.973,Z 164,A -124.2261,B 12.7132,C 0.1573,E1 12.6229,E2 214.3362} C_DIS
LIN {X -72.7082,Y -108.7819,Z 164,A -122.6948,B 12.7132,C 0.1563,E1 12.6265,E2 212.7896} C_DIS
LIN {X -70.0066,Y -110.5401,Z 164,A -121.3278,B 12.7131,C 0.1595,E1 12.6297,E2 211.4282} C_DIS
LIN {X -67.2626,Y -112.2312,Z 164,A -119.8627,B 12.7131,C 0.1602,E1 12.6332,E2 209.957} C_DIS
LIN {X -64.4931,Y -113.8454,Z 164,A -118.5362,B 12.7131,C 0.164,E1 12.6364,E2 208.6398} C_DIS
LIN {X -61.6846,Y -115.391,Z 164,A -117.0164,B 12.7131,C 0.1629,E1 12.6402,E2 207.1064} C_DIS
LIN {X -59.0438,Y -116.7622,Z 164,A -115.6978,B 12.7131,C 0.1641,E1 12.6435,E2 205.786} C_DIS
LIN {X -55.9743,Y -118.2648,Z 164,A -114.2436,B 12.713,C 0.1669,E1 12.6471,E2 204.3369} C_DIS
LIN {X -53.0262,Y -119.6156,Z 164,A -112.7917,B 12.713,C 0.1677,E1 12.6508,E2 202.8812} C_DIS
LIN {X -50.289,Y -120.7912,Z 164,A -111.4498,B 12.713,C 0.1681,E1 12.6543,E2 201.5347} C_DIS
LIN {X -47.0915,Y -122.0737,Z 164,A -109.9068,B 12.713,C 0.1687,E1 12.6583,E2 199.9876} C_DIS
LIN {X -42.7971,Y -123.6443,Z 164,A -107.9606,B 12.713,C 0.1718,E1 12.6634,E2 198.048} C_DIS
LIN {X -39.7542,Y -124.656,Z 164,A -106.5523,B 12.713,C 0.1728,E1 12.6671,E2 196.6391} C_DIS
LIN {X -36.8335,Y -125.55,Z 164,A -105.1425,B 12.713,C 0.172,E1 12.6709,E2 195.2204} C_DIS
LIN {X -33.5864,Y -126.4575,Z 164,A -103.6988,B 12.7129,C 0.1737,E1 12.6748,E2 193.7804} C_DIS
LIN {X -30.6402,Y -127.2034,Z 164,A -102.4447,B 12.7129,C 0.1765,E1 12.6782,E2 192.5353} C_DIS
LIN {X -27.3368,Y -127.9544,Z 164,A -100.8887,B 12.7129,C 0.1754,E1 12.6825,E2 190.9702} C_DIS
LIN {X -24.1914,Y -128.5864,Z 164,A -99.508,B 12.7129,C 0.1766,E1 12.6862,E2 189.5921} C_DIS
LIN {X -21.3588,Y -129.0867,Z 164,A -98.2058,B 12.7129,C 0.1759,E1 12.6898,E2 188.2843} C_DIS
LIN {X -17.6092,Y -129.6528,Z 164,A -96.5667,B 12.7129,C 0.177,E1 12.6944,E2 186.6474} C_DIS
LIN {X -14.4274,Y -130.0447,Z 164,A -95.2389,B 12.7129,C 0.1793,E1 12.698,E2 185.3282} C_DIS
LIN {X -12.0331,Y -130.2882,Z 164,A -93.9449,B 12.7129,C 0.1731,E1 12.7017,E2 184.0049} C_DIS
LIN {X -8.0322,Y -130.5951,Z 164,A -92.4067,B 12.7129,C 0.179,E1 12.7059,E2 182.4923} C_DIS
LIN {X -4.8179,Y -130.7535,Z 164,A -90.9638,B 12.7129,C 0.1781,E1 12.71,E2 181.0448} C_DIS
LIN {X -1.61,Y -130.8333,Z 164,A -89.5811,B 12.7129,C 0.1786,E1 12.7138,E2 179.6642} C_DIS
LIN {X 0.9495,Y -130.8386,Z 164,A -88.9402,B 12.7126,C 0.1911,E1 12.7155,E2 179.0803} C_DIS
Enddeposition()
LIN {X 0.9495,Y -130.8386,Z 164,A -88.9402,B 12.7126,C 0.1911,E1 12.7155,E2 179.0803} C_DIS
Startdeposition()
$VEL.CP = VEL_PRINT
LIN {X -0.8075,Y -131.7592,Z 164,A -89.8661,B 12.7124,C 0.2033,E1 12.7127,E2 180.0615} C_DIS
LIN {X -4.6265,Y -131.6813,Z 164,A -91.4447,B 12.7124,C 0.2012,E1 12.7083,E2 181.6309} C_DIS
LIN {X -8.2381,Y -131.5038,Z 164,A -93.0669,B 12.7124,C 0.2025,E1 12.7037,E2 183.2597} C_DIS
LIN {X -12.4266,Y -131.1743,Z 164,A -94.9434,B 12.7124,C 0.2035,E1 12.6985,E2 185.1428} C_DIS
LIN {X -16.1659,Y -130.7672,Z 164,A -96.4621,B 12.7124,C 0.2002,E1 12.6943,E2 186.6481} C_DIS
LIN {X -18.8446,Y -130.407,Z 164,A -97.6685,B 12.7124,C 0.2007,E1 12.691,E2 187.8586} C_DIS
LIN {X -22.6401,Y -129.803,Z 164,A -99.4853,B 12.7124,C 0.2038,E1 12.6859,E2 189.6933} C_DIS
LIN {X -27.1004,Y -128.9462,Z 164,A -101.2817,B 12.7125,C 0.1984,E1 12.6811,E2 191.4689} C_DIS
LIN {X -30.5085,Y -128.1811,Z 164,A -103.1696,B 12.7124,C 0.207,E1 12.6758,E2 193.4012} C_DIS
LIN {X -33.7048,Y -127.3777,Z 164,A -104.3553,B 12.7124,C 0.1998,E1 12.6727,E2 194.5576} C_DIS
LIN {X -36.9587,Y -126.4716,Z 164,A -106.0636,B 12.7124,C 0.2049,E1 12.668,E2 196.2947} C_DIS
LIN {X -40.0547,Y -125.5254,Z 164,A -107.1928,B 12.7125,C 0.1967,E1 12.6651,E2 197.3908} C_DIS
LIN {X -43.4676,Y -124.3852,Z 164,A -108.7302,B 12.7125,C 0.1947,E1 12.661,E2 198.9251} C_DIS
LIN {X -46.2348,Y -123.3829,Z 164,A -110.1303,B 12.7125,C 0.1966,E1 12.6573,E2 200.3397} C_DIS
LIN {X -49.7648,Y -122.003,Z 164,A -111.6604,B 12.7125,C 0.1921,E1 12.6534,E2 201.8558} C_DIS
LIN {X -52.5482,Y -120.8294,Z 164,A -113.1042,B 12.7125,C 0.194,E1 12.6497,E2 203.3151} C_DIS
LIN {X -55.9205,Y -119.3077,Z 164,A -115.0636,B 12.7125,C 0.2009,E1 12.6446,E2 205.3161} C_DIS
LIN {X -59.4187,Y -117.6033,Z 164,A -116.1453,B 12.7127,C 0.1837,E1 12.6421,E2 206.3251} C_DIS
LIN {X -62.779,Y -115.8465,Z 164,A -117.9377,B 12.7127,C 0.1852,E1 12.6376,E2 208.1346} C_DIS
LIN {X -65.922,Y -114.0868,Z 164,A -119.4901,B 12.7127,C 0.1827,E1 12.6338,E2 209.6851} C_DIS
LIN {X -69.1526,Y -112.1584,Z 164,A -121.3451,B 12.7127,C 0.1858,E1 12.6294,E2 211.5659} C_DIS
LIN {X -73.0217,Y -109.6784,Z 164,A -123.3633,B 12.7127,C 0.1832,E1 12.6246,E2 213.586} C_DIS
LIN {X -76.9596,Y -106.9526,Z 164,A -125.5176,B 12.7127,C 0.1816,E1 12.6197,E2 215.7483} C_DIS
LIN {X -80.8358,Y -104.0532,Z 164,A -128.4954,B 12.7125,C 0.199,E1 12.6129,E2 218.828} C_DIS
LIN {X -86.3791,Y -99.5,Z 164,A -130.6286,B 12.7129,C 0.1698,E1 12.6086,E2 220.8442} C_DIS
LIN {X -89.6224,Y -96.5886,Z 164,A -132.4353,B 12.7129,C 0.164,E1 12.6049,E2 222.6396} C_DIS
LIN {X -92.3231,Y -94.0103,Z 164,A -134.1954,B 12.7129,C 0.164,E1 12.6013,E2 224.4153} C_DIS
LIN {X -95.507,Y -90.7746,Z 164,A -137.1768,B 12.7127,C 0.1838,E1 12.5954,E2 227.5139} C_DIS
LIN {X -100.2868,Y -85.4638,Z 164,A -139.146,B 12.7132,C 0.1504,E1 12.592,E2 229.3481} C_DIS
LIN {X -102.6912,Y -82.5594,Z 164,A -140.8197,B 12.7132,C 0.1475,E1 12.5891,E2 231.0248} C_DIS
LIN {X -104.7637,Y -79.9129,Z 164,A -142.4804,B 12.7132,C 0.1489,E1 12.5862,E2 232.7082} C_DIS
LIN {X -107.4272,Y -76.2958,Z 164,A -144.5312,B 12.7132,C 0.1467,E1 12.5828,E2 234.7693} C_DIS
LIN {X -109.4535,Y -73.3586,Z 164,A -146.0305,B 12.7132,C 0.1417,E1 12.5805,E2 236.2615} C_DIS
LIN {X -112.0686,Y -69.2983,Z 164,A -147.9472,B 12.7133,C 0.1323,E1 12.5776,E2 238.1551} C_DIS
LIN {X -113.5512,Y -66.8404,Z 164,A -149.3854,B 12.7133,C 0.1336,E1 12.5756,E2 239.6147} C_DIS
LIN {X -115.8215,Y -62.8248,Z 164,A -151.474,B 12.7133,C 0.1305,E1 12.5727,E2 241.7116} C_DIS
LIN {X -117.5363,Y -59.5504,Z 164,A -152.9177,B 12.7134,C 0.1225,E1 12.5709,E2 243.1348} C_DIS
LIN {X -119.7849,Y -54.8886,Z 164,A -155.2233,B 12.7134,C 0.1179,E1 12.5681,E2 245.445} C_DIS
LIN {X -121.6231,Y -50.6835,Z 164,A -157.2002,B 12.7135,C 0.1121,E1 12.566,E2 247.418} C_DIS
LIN {X -122.8223,Y -47.7039,Z 164,A -158.691,B 12.7135,C 0.1105,E1 12.5644,E2 248.9187} C_DIS
LIN {X -124.05,Y -44.4147,Z 164,A -160.1784,B 12.7135,C 0.1054,E1 12.563,E2 250.4001} C_DIS
LIN {X -125.0385,Y -41.5497,Z 164,A -161.5088,B 12.7136,C 0.102,E1 12.5618,E2 251.7307} C_DIS
LIN {X -126.1126,Y -38.1678,Z 164,A -163.3228,B 12.7136,C 0.1039,E1 12.5603,E2 253.5751} C_DIS
LIN {X -127.1901,Y -34.4083,Z 164,A -164.8903,B 12.7136,C 0.096,E1 12.5591,E2 255.1255} C_DIS
LIN {X -128.2826,Y -30.0863,Z 164,A -166.8966,B 12.7136,C 0.092,E1 12.5578,E2 257.1379} C_DIS
LIN {X -129.5208,Y -24.2015,Z 164,A -169.3901,B 12.7138,C 0.0817,E1 12.5564,E2 259.6145} C_DIS
LIN {X -130.2891,Y -19.6486,Z 164,A -171.8196,B 12.7138,C 0.0854,E1 12.5553,E2 262.0911} C_DIS
LIN {X -130.777,Y -16.084,Z 164,A -172.8813,B 12.7138,C 0.0695,E1 12.555,E2 263.0925} C_DIS
LIN {X -131.1306,Y -12.8815,Z 164,A -174.4476,B 12.7138,C 0.0691,E1 12.5545,E2 264.6767} C_DIS
LIN {X -131.4456,Y -9.1301,Z 164,A -176.2271,B 12.7138,C 0.0675,E1 12.5541,E2 266.4711} C_DIS
LIN {X -131.6911,Y -4.361,Z 164,A -178.1988,B 12.7138,C 0.059,E1 12.5539,E2 268.4283} C_DIS
LIN {X -131.7597,Y -0.7296,Z 164,A -179.8551,B 12.7139,C 0.056,E1 12.5539,E2 270.0918} C_DIS
LIN {X -131.7296,Y 2.9796,Z 164,A 178.6181,B 12.7139,C 0.0493,E1 12.5539,E2 271.6068} C_DIS
LIN {X -131.6404,Y 5.6756,Z 164,A 177.3532,B 12.7139,C 0.0479,E1 12.554,E2 272.8811} C_DIS
LIN {X -131.4291,Y 9.3564,Z 164,A 175.7374,B 12.7139,C 0.0434,E1 12.5543,E2 274.4965} C_DIS
LIN {X -131.1474,Y 12.7061,Z 164,A 174.238,B 12.7139,C 0.0399,E1 12.5547,E2 275.9986} C_DIS
LIN {X -130.3286,Y 19.3933,Z 164,A 171.3419,B 12.7139,C 0.0306,E1 12.5557,E2 278.8875} C_DIS
LIN {X -129.6738,Y 23.3617,Z 164,A 169.5387,B 12.7139,C 0.0266,E1 12.5566,E2 280.6949} C_DIS
LIN {X -128.9037,Y 27.2973,Z 164,A 167.4588,B 12.7139,C 0.0291,E1 12.5578,E2 282.8117} C_DIS
LIN {X -128.188,Y 30.4801,Z 164,A 166.5122,B 12.714,C 0.0143,E1 12.5583,E2 283.7018} C_DIS
LIN {X -127.5975,Y 32.865,Z 164,A 165.3038,B 12.714,C 0.0143,E1 12.5592,E2 284.9252} C_DIS
LIN {X -126.853,Y 35.628,Z 164,A 164.0273,B 12.714,C 0.0115,E1 12.5601,E2 286.2039} C_DIS
LIN {X -125.9469,Y 38.7093,Z 164,A 162.5376,B 12.714,C 0.0096,E1 12.5613,E2 287.7029} C_DIS
LIN {X -124.8774,Y 42.0336,Z 164,A 160.9234,B 12.714,C 0.0075,E1 12.5627,E2 289.3263} C_DIS
LIN {X -123.3174,Y 46.4097,Z 164,A 159.0015,B 12.714,C -0.0005,E1 12.5646,E2 291.2344} C_DIS
LIN {X -121.8399,Y 50.1642,Z 164,A 156.9693,B 12.714,C 0.001,E1 12.5667,E2 293.2966} C_DIS
LIN {X -120.0349,Y 54.341,Z 164,A 155.236,B 12.714,C -0.01,E1 12.5686,E2 294.9991} C_DIS
LIN {X -118.0879,Y 58.4487,Z 164,A 153.2402,B 12.714,C -0.015,E1 12.5711,E2 296.9947} C_DIS
LIN {X -116.2613,Y 62.0078,Z 164,A 151.3307,B 12.714,C -0.0157,E1 12.5735,E2 298.9219} C_DIS
LIN {X -114.1256,Y 65.8549,Z 164,A 148.5657,B 12.714,C -0.0014,E1 12.5776,E2 301.7823} C_DIS
LIN {X -110.6665,Y 71.5157,Z 164,A 146.6844,B 12.714,C -0.0316,E1 12.5802,E2 303.545} C_DIS
LIN {X -109.2147,Y 73.7134,Z 164,A 145.1685,B 12.714,C -0.026,E1 12.5826,E2 305.1024} C_DIS
LIN {X -107.3766,Y 76.3666,Z 164,A 143.9255,B 12.714,C -0.0331,E1 12.5846,E2 306.3252} C_DIS
LIN {X -104.9173,Y 79.7121,Z 164,A 142.0936,B 12.714,C -0.0369,E1 12.5876,E2 308.1581} C_DIS
LIN {X -102.1221,Y 83.2621,Z 164,A 140.1377,B 12.714,C -0.0417,E1 12.591,E2 310.1106} C_DIS
LIN {X -99.3879,Y 86.5076,Z 164,A 138.2881,B 12.714,C -0.0459,E1 12.5944,E2 311.9587} C_DIS
LIN {X -96.4364,Y 89.7859,Z 164,A 136.3487,B 12.714,C -0.0497,E1 12.5981,E2 313.8982} C_DIS
LIN {X -93.238,Y 93.1036,Z 164,A 134.2963,B 12.714,C -0.0529,E1 12.6021,E2 315.954} C_DIS
LIN {X -90.0555,Y 96.1853,Z 164,A 132.3457,B 12.714,C -0.0564,E1 12.606,E2 317.9053} C_DIS
LIN {X -86.7967,Y 99.1356,Z 164,A 130.4336,B 12.7139,C -0.0603,E1 12.61,E2 319.8154} C_DIS
LIN {X -83.4045,Y 102.0057,Z 164,A 128.5148,B 12.7139,C -0.0644,E1 12.6141,E2 321.7306} C_DIS
LIN {X -80.1268,Y 104.6001,Z 164,A 126.6838,B 12.7139,C -0.0675,E1 12.6181,E2 323.5612} C_DIS
LIN {X -76.775,Y 107.0846,Z 164,A 124.8483,B 12.7139,C -0.0703,E1 12.6223,E2 325.3972} C_DIS
LIN {X -73.3421,Y 109.4645,Z 164,A 123.0039,B 12.7139,C -0.0727,E1 12.6266,E2 327.243} C_DIS
LIN {X -69.629,Y 111.8628,Z 164,A 121.0945,B 12.7139,C -0.0762,E1 12.631,E2 329.149} C_DIS
LIN {X -63.863,Y 115.2519,Z 164,A 118.3844,B 12.7137,C -0.0855,E1 12.6375,E2 331.8335} C_DIS
LIN {X -61.1912,Y 116.6902,Z 164,A 116.9105,B 12.7137,C -0.0837,E1 12.6412,E2 333.324} C_DIS
LIN {X -57.9547,Y 118.3315,Z 164,A 115.268,B 12.7137,C -0.0843,E1 12.6453,E2 334.9725} C_DIS
LIN {X -52.6951,Y 120.7659,Z 164,A 112.9145,B 12.7137,C -0.0916,E1 12.6513,E2 337.3045} C_DIS
LIN {X -50.0667,Y 121.8807,Z 164,A 111.5306,B 12.7137,C -0.0896,E1 12.6549,E2 338.7039} C_DIS
LIN {X -46.2941,Y 123.3607,Z 164,A 109.7402,B 12.7137,C -0.091,E1 12.6595,E2 340.496} C_DIS
LIN {X -42.6513,Y 124.6682,Z 164,A 107.7963,B 12.7137,C -0.0863,E1 12.6647,E2 342.4686} C_DIS
LIN {X -39.6071,Y 125.6684,Z 164,A 106.6926,B 12.7137,C -0.0948,E1 12.6676,E2 343.5379} C_DIS
LIN {X -36.8336,Y 126.5082,Z 164,A 105.3723,B 12.7137,C -0.0945,E1 12.6711,E2 344.8641} C_DIS
LIN {X -33.8189,Y 127.3473,Z 164,A 104.0071,B 12.7137,C -0.0955,E1 12.6748,E2 346.2288} C_DIS
LIN {X -29.8111,Y 128.3455,Z 164,A 102.2216,B 12.7137,C -0.0971,E1 12.6796,E2 348.0119} C_DIS
LIN {X -24.2753,Y 129.5067,Z 164,A 99.8281,B 12.7137,C -0.1004,E1 12.6862,E2 350.396} C_DIS
LIN {X -21.6098,Y 129.9772,Z 164,A 98.628,B 12.7137,C -0.1004,E1 12.6895,E2 351.598} C_DIS
LIN {X -18.3802,Y 130.4734,Z 164,A 97.2592,B 12.7137,C -0.1025,E1 12.6932,E2 352.96} C_DIS
LIN {X -15.2192,Y 130.8801,Z 164,A 95.742,B 12.7137,C -0.0998,E1 12.6975,E2 354.4916} C_DIS
LIN {X -11.4545,Y 131.2632,Z 164,A 94.1647,B 12.7137,C -0.1021,E1 12.7018,E2 356.06} C_DIS
LIN {X -8.2381,Y 131.5038,Z 164,A 92.7389,B 12.7137,C -0.1019,E1 12.7058,E2 357.4877} C_DIS
LIN {X -4.1529,Y 131.697,Z 164,A 90.9139,B 12.7137,C -0.101,E1 12.7109,E2 359.3173} C_DIS
LIN {X 0.0545,Y 131.7633,Z 164,A 89.2087,B 12.7137,C -0.1044,E1 12.7156,E2 361.0072} C_DIS
LIN {X 2.8181,Y 131.7329,Z 164,A 87.9856,B 12.7137,C -0.1038,E1 12.7191,E2 362.2322} C_DIS
LIN {X 5.3172,Y 131.6544,Z 164,A 86.8974,B 12.7137,C -0.1038,E1 12.7221,E2 363.3199} C_DIS
LIN {X 8.6034,Y 131.4813,Z 164,A 85.4564,B 12.7137,C -0.1034,E1 12.7261,E2 364.7616} C_DIS
LIN {X 11.539,Y 131.256,Z 164,A 84.1063,B 12.7137,C -0.1013,E1 12.7299,E2 366.1193} C_DIS
LIN {X 15.6895,Y 130.824,Z 164,A 82.3667,B 12.7137,C -0.1028,E1 12.7347,E2 367.8496} C_DIS
LIN {X 18.8311,Y 130.4089,Z 164,A 80.9653,B 12.7137,C -0.1018,E1 12.7386,E2 369.2532} C_DIS
LIN {X 22.804,Y 129.7737,Z 164,A 79.1858,B 12.7137,C -0.1002,E1 12.7435,E2 371.0357} C_DIS
LIN {X 26.8205,Y 129.0039,Z 164,A 77.1358,B 12.7137,C -0.0922,E1 12.7492,E2 373.1169} C_DIS
LIN {X 30.0127,Y 128.2994,Z 164,A 76.054,B 12.7137,C -0.1003,E1 12.752,E2 374.1589} C_DIS
LIN {X 34.021,Y 127.2934,Z 164,A 73.9416,B 12.7137,C -0.0908,E1 12.7578,E2 376.3076} C_DIS
LIN {X 38.7464,Y 125.9355,Z 164,A 72.053,B 12.7137,C -0.0957,E1 12.7628,E2 378.167} C_DIS
LIN {X 41.9824,Y 124.8944,Z 164,A 70.6703,B 12.7137,C -0.0969,E1 12.7665,E2 379.5385} C_DIS
LIN {X 44.955,Y 123.8552,Z 164,A 69.217,B 12.7137,C -0.0934,E1 12.7703,E2 381.0014} C_DIS
LIN {X 48.0063,Y 122.7048,Z 164,A 67.8454,B 12.7137,C -0.0933,E1 12.7739,E2 382.3676} C_DIS
LIN {X 51.2964,Y 121.3671,Z 164,A 66.1676,B 12.7137,C -0.088,E1 12.7782,E2 384.0609} C_DIS
LIN {X 56.2244,Y 119.1645,Z 164,A 64.0487,B 12.7137,C -0.0914,E1 12.7836,E2 386.1533} C_DIS
LIN {X 58.8379,Y 117.8958,Z 164,A 62.7499,B 12.7137,C -0.0889,E1 12.7868,E2 387.4563} C_DIS
LIN {X 61.6832,Y 116.4319,Z 164,A 61.3762,B 12.7137,C -0.0876,E1 12.7902,E2 388.8281} C_DIS
LIN {X 65.0889,Y 114.5643,Z 164,A 59.6213,B 12.7137,C -0.0834,E1 12.7945,E2 390.5909} C_DIS
LIN {X 67.6632,Y 113.063,Z 164,A 58.3973,B 12.7137,C -0.0835,E1 12.7974,E2 391.8068} C_DIS
LIN {X 70.6622,Y 111.2137,Z 164,A 56.3632,B 12.7139,C -0.0675,E1 12.8024,E2 393.8997} C_DIS
LIN {X 74.1045,Y 108.95,Z 164,A 54.9278,B 12.7139,C -0.0743,E1 12.8056,E2 395.2941} C_DIS
LIN {X 77.32,Y 106.6917,Z 164,A 53.3331,B 12.7139,C -0.0746,E1 12.8092,E2 396.8759} C_DIS
LIN {X 80.5357,Y 104.2858,Z 164,A 51.5158,B 12.7139,C -0.0697,E1 12.8133,E2 398.702} C_DIS
LIN {X 84.1146,Y 101.421,Z 164,A 49.5596,B 12.7139,C -0.0671,E1 12.8175,E2 400.6545} C_DIS
LIN {X 87.5221,Y 98.4961,Z 164,A 47.6456,B 12.7139,C -0.0644,E1 12.8215,E2 402.5647} C_DIS
LIN {X 90.609,Y 95.6638,Z 164,A 45.8501,B 12.7139,C -0.0616,E1 12.8252,E2 404.3579} C_DIS
LIN {X 93.5259,Y 92.8138,Z 164,A 44.0944,B 12.7139,C -0.0585,E1 12.8287,E2 406.1124} C_DIS
LIN {X 96.4356,Y 89.7867,Z 164,A 42.2707,B 12.7139,C -0.0547,E1 12.8322,E2 407.9367} C_DIS
LIN {X 99.3404,Y 86.562,Z 164,A 40.3825,B 12.7139,C -0.0506,E1 12.8357,E2 409.8259} C_DIS
LIN {X 102.2321,Y 83.1276,Z 164,A 38.486,B 12.7139,C -0.0478,E1 12.839,E2 411.717} C_DIS
LIN {X 104.5376,Y 80.2086,Z 164,A 36.8573,B 12.7139,C -0.0438,E1 12.8418,E2 413.348} C_DIS
LIN {X 106.7909,Y 77.183,Z 164,A 35.2276,B 12.7139,C -0.0402,E1 12.8445,E2 414.9775} C_DIS
LIN {X 108.9517,Y 74.102,Z 164,A 33.5518,B 12.7139,C -0.0352,E1 12.8472,E2 416.6589} C_DIS
LIN {X 111.2023,Y 70.6804,Z 164,A 31.811,B 12.7139,C -0.032,E1 12.8498,E2 418.3962} C_DIS
LIN {X 113.7871,Y 66.4387,Z 164,A 29.7204,B 12.7139,C -0.0285,E1 12.8528,E2 420.4802} C_DIS
LIN {X 115.8213,Y 62.8253,Z 164,A 27.8838,B 12.714,C -0.023,E1 12.8553,E2 422.3221} C_DIS
LIN {X 117.6587,Y 59.3099,Z 164,A 26.2321,B 12.714,C -0.0206,E1 12.8574,E2 423.9665} C_DIS
LIN {X 119.2049,Y 56.1399,Z 164,A 24.7871,B 12.714,C -0.0191,E1 12.8591,E2 425.4022} C_DIS
LIN {X 120.3571,Y 53.6207,Z 164,A 23.6013,B 12.714,C -0.0164,E1 12.8605,E2 426.5868} C_DIS
LIN {X 121.6934,Y 50.5152,Z 164,A 22.1099,B 12.714,C -0.0118,E1 12.8621,E2 428.0819} C_DIS
LIN {X 122.8805,Y 47.5543,Z 164,A 20.7157,B 12.714,C -0.0078,E1 12.8635,E2 429.4782} C_DIS
LIN {X 124.1564,Y 44.1197,Z 164,A 19.0395,B 12.714,C -0.001,E1 12.8652,E2 431.1657} C_DIS
LIN {X 125.7189,Y 39.447,Z 164,A 16.7914,B 12.714,C 0.008,E1 12.8671,E2 433.4282} C_DIS
LIN {X 127.6659,Y 32.5955,Z 164,A 13.9343,B 12.714,C 0.0098,E1 12.8692,E2 436.2597} C_DIS
LIN {X 128.6491,Y 28.4767,Z 164,A 12.2333,B 12.714,C 0.0111,E1 12.8703,E2 437.946} C_DIS
LIN {X 129.1843,Y 25.9342,Z 164,A 11.0763,B 12.714,C 0.0151,E1 12.8709,E2 439.1073} C_DIS
LIN {X 129.8898,Y 22.134,Z 164,A 9.2756,B 12.714,C 0.0235,E1 12.8718,E2 440.9239} C_DIS
LIN {X 130.5166,Y 18.0781,Z 164,A 7.4963,B 12.714,C 0.0286,E1 12.8725,E2 442.7044} C_DIS
LIN {X 131.0033,Y 14.1143,Z 164,A 5.8505,B 12.714,C 0.031,E1 12.873,E2 444.3413} C_DIS
LIN {X 131.3207,Y 10.7731,Z 164,A 4.3846,B 12.714,C 0.0355,E1 12.8734,E2 445.8095} C_DIS
LIN {X 131.5898,Y 6.7271,Z 164,A 2.7,B 12.714,C 0.0384,E1 12.8737,E2 447.4867} C_DIS
LIN {X 131.7319,Y 2.8789,Z 164,A 0.9523,B 12.714,C 0.0456,E1 12.8738,E2 449.245} C_DIS
LIN {X 131.756,Y -1.4013,Z 164,A -0.7238,B 12.714,C 0.0456,E1 12.8738,E2 450.9012} C_DIS
LIN {X 131.6957,Y -4.1994,Z 164,A -2.0625,B 12.714,C 0.0528,E1 12.8738,E2 452.2557} C_DIS
LIN {X 131.5037,Y -8.2406,Z 164,A -3.6499,B 12.714,C 0.053,E1 12.8735,E2 453.8246} C_DIS
LIN {X 131.2792,Y -11.2641,Z 164,A -5.0235,B 12.7139,C 0.0586,E1 12.8732,E2 455.2063} C_DIS
LIN {X 130.9815,Y -14.3174,Z 164,A -6.3132,B 12.7139,C 0.0612,E1 12.8728,E2 456.4923} C_DIS
LIN {X 130.4912,Y -18.2554,Z 164,A -8.0853,B 12.7139,C 0.0677,E1 12.8721,E2 458.272} C_DIS
LIN {X 129.8528,Y -22.3552,Z 164,A -9.9352,B 12.7139,C 0.0744,E1 12.8713,E2 460.1295} C_DIS
LIN {X 129.0039,Y -26.8208,Z 164,A -11.7438,B 12.7139,C 0.0753,E1 12.8703,E2 461.9204} C_DIS
LIN {X 127.9091,Y -31.6369,Z 164,A -13.8672,B 12.7138,C 0.0808,E1 12.869,E2 464.0435} C_DIS
LIN {X 126.6973,Y -36.1846,Z 164,A -15.8845,B 12.7138,C 0.0859,E1 12.8675,E2 466.0597} C_DIS
LIN {X 125.8304,Y -39.0901,Z 164,A -17.2564,B 12.7138,C 0.0913,E1 12.8664,E2 467.4396} C_DIS
LIN {X 124.4688,Y -43.2263,Z 164,A -18.9947,B 12.7137,C 0.0921,E1 12.8649,E2 469.1615} C_DIS
LIN {X 123.5532,Y -45.78,Z 164,A -20.3356,B 12.7137,C 0.1002,E1 12.8635,E2 470.5232} C_DIS
LIN {X 122.1473,Y -49.407,Z 164,A -21.9296,B 12.7137,C 0.1021,E1 12.8619,E2 472.1075} C_DIS
LIN {X 120.6484,Y -52.9669,Z 164,A -23.7194,B 12.7136,C 0.11,E1 12.8599,E2 473.9127} C_DIS
LIN {X 117.2804,Y -60.0531,Z 164,A -26.9695,B 12.7136,C 0.1146,E1 12.856,E2 477.1476} C_DIS
LIN {X 115.6039,Y -63.2237,Z 164,A -28.9375,B 12.7134,C 0.1306,E1 12.8533,E2 479.1663} C_DIS
LIN {X 113.6635,Y -66.6492,Z 164,A -30.0938,B 12.7134,C 0.119,E1 12.8518,E2 480.2582} C_DIS
LIN {X 112.3123,Y -68.9016,Z 164,A -31.3334,B 12.7134,C 0.1248,E1 12.85,E2 481.5109} C_DIS
LIN {X 110.5211,Y -71.7396,Z 164,A -32.8511,B 12.7134,C 0.1303,E1 12.8477,E2 483.0374} C_DIS
LIN {X 108.1437,Y -75.2756,Z 164,A -34.6296,B 12.7134,C 0.1328,E1 12.8449,E2 484.8092} C_DIS
LIN {X 105.8169,Y -78.5132,Z 164,A -36.3102,B 12.7134,C 0.1355,E1 12.8421,E2 486.4854} C_DIS
LIN {X 103.566,Y -81.459,Z 164,A -37.969,B 12.7133,C 0.1408,E1 12.8393,E2 488.1518} C_DIS
LIN {X 100.767,Y -84.8974,Z 164,A -39.749,B 12.7133,C 0.1411,E1 12.8361,E2 489.9163} C_DIS
LIN {X 98.8533,Y -87.118,Z 164,A -41.1856,B 12.7132,C 0.1487,E1 12.8335,E2 491.3738} C_DIS
LIN {X 95.9099,Y -90.3482,Z 164,A -43.0076,B 12.7132,C 0.1508,E1 12.83,E2 493.1886} C_DIS
LIN {X 93.1224,Y -93.2186,Z 164,A -44.743,B 12.7132,C 0.1545,E1 12.8266,E2 494.9254} C_DIS
LIN {X 90.8446,Y -95.4401,Z 164,A -46.159,B 12.7131,C 0.1584,E1 12.8238,E2 496.3468} C_DIS
LIN {X 87.8566,Y -98.1973,Z 164,A -47.9192,B 12.7131,C 0.1619,E1 12.8201,E2 498.1081} C_DIS
LIN {X 84.7657,Y -100.8775,Z 164,A -49.667,B 12.713,C 0.1646,E1 12.8164,E2 499.8541} C_DIS
LIN {X 82.0527,Y -103.0962,Z 164,A -51.0149,B 12.713,C 0.1626,E1 12.8135,E2 501.1824} C_DIS
LIN {X 79.457,Y -105.1099,Z 164,A -52.6585,B 12.7129,C 0.1715,E1 12.8098,E2 502.8535} C_DIS
LIN {X 75.9327,Y -107.6834,Z 164,A -54.2997,B 12.7129,C 0.1677,E1 12.8062,E2 504.4657} C_DIS
LIN {X 72.9188,Y -109.7471,Z 164,A -56.099,B 12.7129,C 0.1765,E1 12.8019,E2 506.292} C_DIS
LIN {X 70.0232,Y -111.6171,Z 164,A -57.4643,B 12.7129,C 0.1753,E1 12.7988,E2 507.6429} C_DIS
LIN {X 67.2505,Y -113.309,Z 164,A -58.9785,B 12.7128,C 0.1805,E1 12.7951,E2 509.1706} C_DIS
LIN {X 64.0044,Y -115.1737,Z 164,A -60.4639,B 12.7128,C 0.1791,E1 12.7915,E2 510.6405} C_DIS
LIN {X 61.074,Y -116.7517,Z 164,A -61.9667,B 12.7128,C 0.1828,E1 12.7878,E2 512.1514} C_DIS
LIN {X 57.9995,Y -118.3095,Z 164,A -63.398,B 12.7128,C 0.1831,E1 12.7842,E2 513.5759} C_DIS
LIN {X 55.1749,Y -119.6525,Z 164,A -64.7839,B 12.7127,C 0.1857,E1 12.7807,E2 514.9661} C_DIS
LIN {X 51.4351,Y -121.3092,Z 164,A -66.6943,B 12.7127,C 0.1917,E1 12.7758,E2 516.8941} C_DIS
LIN {X 47.0516,Y -123.0759,Z 164,A -68.5657,B 12.7127,C 0.1891,E1 12.771,E2 518.7452} C_DIS
LIN {X 43.9121,Y -124.2311,Z 164,A -70.2867,B 12.7125,C 0.1981,E1 12.7664,E2 520.4993} C_DIS
LIN {X 39.2975,Y -125.7669,Z 164,A -72.1092,B 12.7125,C 0.1923,E1 12.7616,E2 522.2884} C_DIS
LIN {X 31.6568,Y -127.9042,Z 164,A -75.5373,B 12.7125,C 0.1949,E1 12.7524,E2 525.7167} C_DIS
LIN {X 26.628,Y -129.0431,Z 164,A -77.9453,B 12.7125,C 0.2011,E1 12.7457,E2 528.1462} C_DIS
LIN {X 22.4892,Y -129.83,Z 164,A -79.6069,B 12.7125,C 0.1978,E1 12.7412,E2 529.7886} C_DIS
LIN {X 19.6926,Y -130.2823,Z 164,A -80.8326,B 12.7125,C 0.1983,E1 12.7379,E2 531.0142} C_DIS
LIN {X 16.151,Y -130.769,Z 164,A -82.4995,B 12.7125,C 0.2022,E1 12.7332,E2 532.6956} C_DIS
LIN {X 12.3453,Y -131.1821,Z 164,A -84.0215,B 12.7125,C 0.1991,E1 12.729,E2 534.2014} C_DIS
LIN {X 9.2378,Y -131.4378,Z 164,A -85.5577,B 12.7125,C 0.2044,E1 12.7247,E2 535.7601} C_DIS
LIN {X 5.1071,Y -131.6625,Z 164,A -87.2197,B 12.7125,C 0.2012,E1 12.7201,E2 537.4067} C_DIS
LIN {X 1.8384,Y -131.7492,Z 164,A -88.5901,B 12.7125,C 0.2002,E1 12.7163,E2 538.7716} C_DIS
LIN {X 1.8384,Y -131.7492,Z 164,A -88.5901,B 12.7125,C 0.2002,E1 12.7163,E2 538.7716} C_DIS
Enddeposition()
LIN {X 0.9686,Y -132.6764,Z 164,A -88.4296,B 12.7125,C 0.1936,E1 12.7168,E2 538.5813} C_DIS
Startdeposition()
$VEL.CP = VEL_PRINT
LIN {X 4.449,Y -132.6086,Z 164,A -86.7814,B 12.7126,C 0.1894,E1 12.7215,E2 536.9146} C_DIS
LIN {X 8.1366,Y -132.4314,Z 164,A -85.3124,B 12.7126,C 0.1923,E1 12.7255,E2 535.4601} C_DIS
LIN {X 10.7965,Y -132.2417,Z 164,A -84.0712,B 12.7126,C 0.1894,E1 12.729,E2 534.2072} C_DIS
LIN {X 13.8887,Y -131.9525,Z 164,A -82.749,B 12.7126,C 0.1894,E1 12.7327,E2 532.8866} C_DIS
LIN {X 17.4947,Y -131.5229,Z 164,A -81.1331,B 12.7126,C 0.1872,E1 12.7372,E2 531.2638} C_DIS
LIN {X 21.5879,Y -130.9132,Z 164,A -79.4269,B 12.7126,C 0.1884,E1 12.7418,E2 529.5664} C_DIS
LIN {X 24.8648,Y -130.3303,Z 164,A -78.0422,B 12.7126,C 0.1889,E1 12.7456,E2 528.1871} C_DIS
LIN {X 27.6929,Y -129.7591,Z 164,A -76.5465,B 12.7128,C 0.181,E1 12.7498,E2 526.6599} C_DIS
LIN {X 31.9395,Y -128.7812,Z 164,A -74.4806,B 12.7128,C 0.1743,E1 12.7555,E2 524.57} C_DIS
LIN {X 35.3971,Y -127.8724,Z 164,A -72.9766,B 12.7128,C 0.174,E1 12.7595,E2 523.0697} C_DIS
LIN {X 38.7503,Y -126.8961,Z 164,A -72.0595,B 12.7126,C 0.189,E1 12.7618,E2 522.224} C_DIS
LIN {X 43.9971,Y -125.1749,Z 164,A -69.4426,B 12.7128,C 0.18,E1 12.7688,E2 519.5769} C_DIS
LIN {X 47.4138,Y -123.9218,Z 164,A -67.8385,B 12.7128,C 0.1772,E1 12.773,E2 517.9675} C_DIS
LIN {X 50.8078,Y -122.5678,Z 164,A -66.2683,B 12.7128,C 0.1755,E1 12.7771,E2 516.3968} C_DIS
LIN {X 53.978,Y -121.2047,Z 164,A -64.7394,B 12.7128,C 0.1724,E1 12.781,E2 514.8618} C_DIS
LIN {X 57.8773,Y -119.3941,Z 164,A -62.8451,B 12.7129,C 0.1687,E1 12.7858,E2 512.9613} C_DIS
LIN {X 61.659,Y -117.4833,Z 164,A -61.2412,B 12.7129,C 0.1724,E1 12.7897,E2 511.3833} C_DIS
LIN {X 64.9419,Y -115.7032,Z 164,A -59.4959,B 12.7129,C 0.1662,E1 12.794,E2 509.6202} C_DIS
LIN {X 68.5856,Y -113.5813,Z 164,A -57.6503,B 12.713,C 0.1625,E1 12.7984,E2 507.7698} C_DIS
LIN {X 74.2887,Y -109.9358,Z 164,A -54.8396,B 12.713,C 0.1607,E1 12.805,E2 504.9699} C_DIS
LIN {X 77.3031,Y -107.8376,Z 164,A -53.164,B 12.713,C 0.1552,E1 12.8089,E2 503.2818} C_DIS
LIN {X 81.0039,Y -105.0865,Z 164,A -51.103,B 12.7132,C 0.1494,E1 12.8135,E2 501.21} C_DIS
LIN {X 85.8972,Y -101.1254,Z 164,A -48.5568,B 12.7132,C 0.149,E1 12.8189,E2 498.6821} C_DIS
LIN {X 88.8807,Y -98.5141,Z 164,A -46.8123,B 12.7132,C 0.1445,E1 12.8226,E2 496.9318} C_DIS
LIN {X 93.081,Y -94.5551,Z 164,A -44.0786,B 12.7134,C 0.132,E1 12.8281,E2 494.1655} C_DIS
LIN {X 95.6102,Y -91.9974,Z 164,A -42.7835,B 12.7134,C 0.1362,E1 12.8306,E2 492.9005} C_DIS
LIN {X 98.5663,Y -88.823,Z 164,A -40.976,B 12.7134,C 0.1338,E1 12.834,E2 491.0989} C_DIS
LIN {X 102.2004,Y -84.6153,Z 164,A -38.5962,B 12.7134,C 0.1288,E1 12.8383,E2 488.7189} C_DIS
LIN {X 105.0164,Y -81.0944,Z 164,A -36.6169,B 12.7134,C 0.1231,E1 12.8417,E2 486.7334} C_DIS
LIN {X 107.4561,Y -77.8323,Z 164,A -34.9184,B 12.7134,C 0.1206,E1 12.8445,E2 485.0402} C_DIS
LIN {X 109.9264,Y -74.3027,Z 164,A -33.1147,B 12.7134,C 0.1176,E1 12.8473,E2 483.2412} C_DIS
LIN {X 112.1453,Y -70.9093,Z 164,A -31.3504,B 12.7135,C 0.1127,E1 12.85,E2 481.4731} C_DIS
LIN {X 114.1637,Y -67.6127,Z 164,A -29.6006,B 12.7135,C 0.1059,E1 12.8525,E2 479.7115} C_DIS
LIN {X 116.7441,Y -63.0523,Z 164,A -27.4342,B 12.7136,C 0.1028,E1 12.8555,E2 477.5541} C_DIS
LIN {X 119.1533,Y -58.3676,Z 164,A -24.9452,B 12.7137,C 0.0902,E1 12.8586,E2 475.036} C_DIS
LIN {X 120.6429,Y -55.2241,Z 164,A -23.6871,B 12.7137,C 0.0934,E1 12.8601,E2 473.8061} C_DIS
LIN {X 122.1931,Y -51.705,Z 164,A -22.0773,B 12.7137,C 0.0903,E1 12.8618,E2 472.2005} C_DIS
LIN {X 123.398,Y -48.7612,Z 164,A -20.5069,B 12.7137,C 0.0805,E1 12.8635,E2 470.6043} C_DIS
LIN {X 124.5455,Y -45.7519,Z 164,A -19.3204,B 12.7137,C 0.0827,E1 12.8646,E2 469.4411} C_DIS
LIN {X 126.7343,Y -39.2789,Z 164,A -16.4392,B 12.7137,C 0.0763,E1 12.8671,E2 466.5649} C_DIS
LIN {X 127.7919,Y -35.6852,Z 164,A -14.3609,B 12.7139,C 0.0579,E1 12.8687,E2 464.4281} C_DIS
LIN {X 128.9386,Y -31.2904,Z 164,A -12.8778,B 12.7139,C 0.0665,E1 12.8697,E2 463.0014} C_DIS
LIN {X 129.8516,Y -27.2647,Z 164,A -11.0321,B 12.7139,C 0.0594,E1 12.8708,E2 461.146} C_DIS
LIN {X 130.5658,Y -23.5978,Z 164,A -9.5298,B 12.7139,C 0.058,E1 12.8715,E2 459.6552} C_DIS
LIN {X 131.2827,Y -19.2175,Z 164,A -7.6444,B 12.7139,C 0.0532,E1 12.8723,E2 457.7714} C_DIS
LIN {X 131.8258,Y -15.0554,Z 164,A -5.9082,B 12.7139,C 0.0502,E1 12.8729,E2 456.0424} C_DIS
LIN {X 132.2091,Y -11.182,Z 164,A -4.2323,B 12.7139,C 0.0453,E1 12.8734,E2 454.3651} C_DIS
LIN {X 132.4911,Y -7.1147,Z 164,A -2.4598,B 12.7139,C 0.0397,E1 12.8737,E2 452.5892} C_DIS
LIN {X 132.6317,Y -3.6265,Z 164,A -0.998,B 12.7139,C 0.0366,E1 12.8737,E2 451.1312} C_DIS
LIN {X 132.6807,Y 0.4739,Z 164,A 0.6716,B 12.7139,C 0.0343,E1 12.8738,E2 449.4719} C_DIS
LIN {X 132.6215,Y 3.993,Z 164,A 2.2318,B 12.7139,C 0.0286,E1 12.8738,E2 447.9051} C_DIS
LIN {X 132.44,Y 7.9978,Z 164,A 3.975,B 12.714,C 0.0231,E1 12.8735,E2 446.1586} C_DIS
LIN {X 132.1637,Y 11.7196,Z 164,A 5.6498,B 12.714,C 0.0165,E1 12.8731,E2 444.4744} C_DIS
LIN {X 131.7567,Y 15.6348,Z 164,A 7.2014,B 12.714,C 0.0159,E1 12.8726,E2 442.9389} C_DIS
LIN {X 131.257,Y 19.3974,Z 164,A 8.9186,B 12.714,C 0.0088,E1 12.8719,E2 441.2106} C_DIS
LIN {X 130.6202,Y 23.2943,Z 164,A 10.479,B 12.714,C 0.0081,E1 12.8712,E2 439.666} C_DIS
LIN {X 129.9784,Y 26.6437,Z 164,A 11.9581,B 12.714,C 0.0037,E1 12.8704,E2 438.1846} C_DIS
LIN {X 129.1362,Y 30.4708,Z 164,A 13.7166,B 12.714,C -0.0032,E1 12.8693,E2 436.4165} C_DIS
LIN {X 127.565,Y 36.4897,Z 164,A 16.2144,B 12.714,C -0.0052,E1 12.8675,E2 433.939} C_DIS
LIN {X 125.6408,Y 42.6517,Z 164,A 19.0593,B 12.714,C -0.0147,E1 12.8651,E2 431.0847} C_DIS
LIN {X 124.539,Y 45.7683,Z 164,A 20.4763,B 12.714,C -0.0183,E1 12.8637,E2 429.6677} C_DIS
LIN {X 123.3691,Y 48.8355,Z 164,A 21.9796,B 12.714,C -0.0247,E1 12.8622,E2 428.1528} C_DIS
LIN {X 121.9303,Y 52.3193,Z 164,A 23.5594,B 12.714,C -0.0277,E1 12.8605,E2 426.5774} C_DIS
LIN {X 120.4921,Y 55.5503,Z 164,A 24.985,B 12.714,C -0.0288,E1 12.8588,E2 425.1628} C_DIS
LIN {X 117.7558,Y 61.14,Z 164,A 27.729,B 12.714,C -0.0375,E1 12.8554,E2 422.41} C_DIS
LIN {X 115.9978,Y 64.4145,Z 164,A 29.7376,B 12.714,C -0.0534,E1 12.8526,E2 420.3513} C_DIS
LIN {X 113.8236,Y 68.1832,Z 164,A 31.1749,B 12.714,C -0.0452,E1 12.8507,E2 418.9662} C_DIS
LIN {X 111.5649,Y 71.8196,Z 164,A 33.001,B 12.714,C -0.0491,E1 12.8479,E2 417.1414} C_DIS
LIN {X 109.7669,Y 74.5382,Z 164,A 34.5468,B 12.714,C -0.0565,E1 12.8455,E2 415.5781} C_DIS
LIN {X 106.832,Y 78.6869,Z 164,A 36.5909,B 12.7139,C -0.0573,E1 12.8422,E2 413.5507} C_DIS
LIN {X 104.0885,Y 82.2826,Z 164,A 38.5497,B 12.7139,C -0.062,E1 12.8388,E2 411.5901} C_DIS
LIN {X 101.2613,Y 85.7373,Z 164,A 40.4501,B 12.7139,C -0.0655,E1 12.8354,E2 409.6919} C_DIS
LIN {X 98.3547,Y 89.0565,Z 164,A 42.3262,B 12.7139,C -0.0688,E1 12.8319,E2 407.8182} C_DIS
LIN {X 95.3646,Y 92.2512,Z 164,A 44.194,B 12.7139,C -0.0721,E1 12.8283,E2 405.9522} C_DIS
LIN {X 92.1513,Y 95.4613,Z 164,A 46.1295,B 12.7139,C -0.0754,E1 12.8245,E2 404.0189} C_DIS
LIN {X 88.8952,Y 98.501,Z 164,A 48.0655,B 12.7138,C -0.0795,E1 12.8205,E2 402.0807} C_DIS
LIN {X 85.5439,Y 101.425,Z 164,A 49.9529,B 12.7138,C -0.0821,E1 12.8165,E2 400.1965} C_DIS
LIN {X 82.288,Y 104.0842,Z 164,A 51.7935,B 12.7138,C -0.0861,E1 12.8125,E2 398.3523} C_DIS
LIN {X 78.7325,Y 106.7985,Z 164,A 53.6883,B 12.7138,C -0.0884,E1 12.8083,E2 396.4613} C_DIS
LIN {X 74.9774,Y 109.4673,Z 164,A 55.7134,B 12.7137,C -0.0926,E1 12.8036,E2 394.4314} C_DIS
LIN {X 71.0577,Y 112.0516,Z 164,A 57.6935,B 12.7137,C -0.0944,E1 12.799,E2 392.4567} C_DIS
LIN {X 67.6127,Y 114.1637,Z 164,A 59.6284,B 12.7137,C -0.1023,E1 12.7943,E2 390.4987} C_DIS
LIN {X 64.6856,Y 115.8473,Z 164,A 60.8702,B 12.7137,C -0.0983,E1 12.7913,E2 389.2826} C_DIS
LIN {X 60.5661,Y 118.0512,Z 164,A 62.9412,B 12.7137,C -0.1024,E1 12.7862,E2 387.205} C_DIS
LIN {X 57.0588,Y 119.7851,Z 164,A 64.5813,B 12.7137,C -0.1031,E1 12.7821,E2 385.5706} C_DIS
LIN {X 53.0377,Y 121.6197,Z 164,A 66.3631,B 12.7137,C -0.1018,E1 12.7776,E2 383.804} C_DIS
LIN {X 50.3225,Y 122.7698,Z 164,A 67.7179,B 12.7136,C -0.1054,E1 12.7741,E2 382.4395} C_DIS
LIN {X 46.8335,Y 124.1407,Z 164,A 69.1041,B 12.7136,C -0.1007,E1 12.7705,E2 381.081} C_DIS
LIN {X 43.6124,Y 125.3083,Z 164,A 70.7116,B 12.7136,C -0.1055,E1 12.7662,E2 379.4584} C_DIS
LIN {X 40.7528,Y 126.2678,Z 164,A 72.0094,B 12.7136,C -0.1065,E1 12.7628,E2 378.1613} C_DIS
LIN {X 34.5436,Y 128.1058,Z 164,A 74.7096,B 12.7136,C -0.106,E1 12.7556,E2 375.473} C_DIS
LIN {X 28.0819,Y 129.6751,Z 164,A 77.7201,B 12.7136,C -0.1115,E1 12.7474,E2 372.4466} C_DIS
LIN {X 23.7045,Y 130.5467,Z 164,A 79.601,B 12.7136,C -0.1112,E1 12.7422,E2 370.5717} C_DIS
LIN {X 20.6197,Y 131.0694,Z 164,A 80.9779,B 12.7136,C -0.1124,E1 12.7384,E2 369.1922} C_DIS
LIN {X 16.9852,Y 131.5896,Z 164,A 82.5953,B 12.7136,C -0.1138,E1 12.7339,E2 367.5715} C_DIS
LIN {X 13.255,Y 132.0186,Z 164,A 84.2122,B 12.7136,C -0.1141,E1 12.7294,E2 365.9557} C_DIS
LIN {X 9.7233,Y 132.3244,Z 164,A 85.665,B 12.7136,C -0.1123,E1 12.7254,E2 364.5127} C_DIS
LIN {X 6.0981,Y 132.5422,Z 164,A 87.3335,B 12.7136,C -0.115,E1 12.7207,E2 362.8331} C_DIS
LIN {X 2.3945,Y 132.6598,Z 164,A 88.8786,B 12.7136,C -0.1136,E1 12.7164,E2 361.2952} C_DIS
LIN {X -1.8914,Y 132.6681,Z 164,A 90.7145,B 12.7136,C -0.1131,E1 12.7113,E2 359.4619} C_DIS
LIN {X -5.3796,Y 132.5723,Z 164,A 92.1829,B 12.7136,C -0.1118,E1 12.7072,E2 357.9988} C_DIS
LIN {X -9.0899,Y 132.3706,Z 164,A 93.8799,B 12.7136,C -0.1138,E1 12.7025,E2 356.2918} C_DIS
LIN {X -13.223,Y 132.0217,Z 164,A 95.6101,B 12.7136,C -0.1116,E1 12.6977,E2 354.5698} C_DIS
LIN {X -17.2205,Y 131.5588,Z 164,A 97.2504,B 12.7136,C -0.1084,E1 12.6932,E2 352.942} C_DIS
LIN {X -20.4462,Y 131.0963,Z 164,A 98.7577,B 12.7136,C -0.1102,E1 12.689,E2 351.4237} C_DIS
LIN {X -24.3678,Y 130.4253,Z 164,A 101.5235,B 12.7133,C -0.1361,E1 12.6811,E2 348.534} C_DIS
LIN {X -31.3953,Y 128.9133,Z 164,A 103.6243,B 12.7136,C -0.1081,E1 12.6757,E2 346.5554} C_DIS
LIN {X -35.5011,Y 127.8434,Z 164,A 105.2926,B 12.7136,C -0.1024,E1 12.6712,E2 344.9078} C_DIS
LIN {X -42.3519,Y 125.7407,Z 164,A 108.514,B 12.7136,C -0.1026,E1 12.6626,E2 341.674} C_DIS
LIN {X -45.7908,Y 124.5312,Z 164,A 110.171,B 12.7136,C -0.103,E1 12.6582,E2 340.0086} C_DIS
LIN {X -49.3864,Y 123.1471,Z 164,A 111.7372,B 12.7136,C -0.0986,E1 12.6542,E2 338.4553} C_DIS
LIN {X -52.3737,Y 121.9068,Z 164,A 114.1575,B 12.7134,C -0.1225,E1 12.6477,E2 335.9142} C_DIS
LIN {X -58.5265,Y 119.0749,Z 164,A 115.9095,B 12.7137,C -0.0893,E1 12.6437,E2 334.3047} C_DIS
LIN {X -65.4721,Y 115.4045,Z 164,A 119.6054,B 12.7137,C -0.0917,E1 12.6345,E2 330.5764} C_DIS
LIN {X -69.0818,Y 113.2807,Z 164,A 121.4755,B 12.7137,C -0.0904,E1 12.63,E2 328.7008} C_DIS
LIN {X -72.8431,Y 110.899,Z 164,A 123.3646,B 12.7137,C -0.0864,E1 12.6256,E2 326.8176} C_DIS
LIN {X -76.128,Y 108.671,Z 164,A 125.1226,B 12.7137,C -0.0844,E1 12.6215,E2 325.0561} C_DIS
LIN {X -79.7018,Y 106.0772,Z 164,A 127.0491,B 12.7137,C -0.0814,E1 12.6172,E2 323.1293} C_DIS
LIN {X -83.3379,Y 103.2447,Z 164,A 129.0091,B 12.7137,C -0.0769,E1 12.6129,E2 321.175} C_DIS
LIN {X -86.669,Y 100.4648,Z 164,A 130.9133,B 12.7138,C -0.0739,E1 12.6089,E2 319.2692} C_DIS
LIN {X -90.0758,Y 97.4227,Z 164,A 132.929,B 12.7138,C -0.0709,E1 12.6047,E2 317.2505} C_DIS
LIN {X -93.1205,Y 94.5164,Z 164,A 134.7338,B 12.7138,C -0.0668,E1 12.6011,E2 315.4493} C_DIS
LIN {X -96.0464,Y 91.5413,Z 164,A 136.4967,B 12.7138,C -0.0619,E1 12.5977,E2 313.693} C_DIS
LIN {X -98.8163,Y 88.5439,Z 164,A 138.3403,B 12.7138,C -0.0599,E1 12.5942,E2 311.8418} C_DIS
LIN {X -101.6677,Y 85.2547,Z 164,A 140.2102,B 12.7139,C -0.0553,E1 12.5908,E2 309.9752} C_DIS
LIN {X -104.4564,Y 81.8142,Z 164,A 142.1312,B 12.7139,C -0.051,E1 12.5875,E2 308.0554} C_DIS
LIN {X -107.1256,Y 78.2873,Z 164,A 143.9823,B 12.7139,C -0.0449,E1 12.5844,E2 306.2136} C_DIS
LIN {X -108.565,Y 76.278,Z 164,A 145.1716,B 12.7139,C -0.0452,E1 12.5825,E2 305.0111} C_DIS
LIN {X -110.8975,Y 72.8454,Z 164,A 147.4151,B 12.7139,C -0.0513,E1 12.5789,E2 302.716} C_DIS
LIN {X -113.2337,Y 69.1573,Z 164,A 148.9016,B 12.7139,C -0.0371,E1 12.5768,E2 301.2793} C_DIS
LIN {X -116.2876,Y 63.8908,Z 164,A 151.4834,B 12.7139,C -0.029,E1 12.5733,E2 298.7063} C_DIS
LIN {X -118.0653,Y 60.5383,Z 164,A 152.9285,B 12.714,C -0.0202,E1 12.5714,E2 297.286} C_DIS
LIN {X -120.4579,Y 55.6243,Z 164,A 155.983,B 12.714,C -0.03,E1 12.5677,E2 294.1519} C_DIS
LIN {X -122.1928,Y 51.7057,Z 164,A 157.422,B 12.714,C -0.0152,E1 12.5661,E2 292.7643} C_DIS
LIN {X -123.5753,Y 48.3052,Z 164,A 158.9575,B 12.714,C -0.0097,E1 12.5646,E2 291.2365} C_DIS
LIN {X -124.8963,Y 44.779,Z 164,A 160.638,B 12.714,C -0.0063,E1 12.5629,E2 289.5515} C_DIS
LIN {X -126.2713,Y 40.7418,Z 164,A 162.4604,B 12.714,C -0.0007,E1 12.5613,E2 287.7337} C_DIS
Enddeposition()
END
